Yaskawa INFORM job: test_long_tjr4.JBI

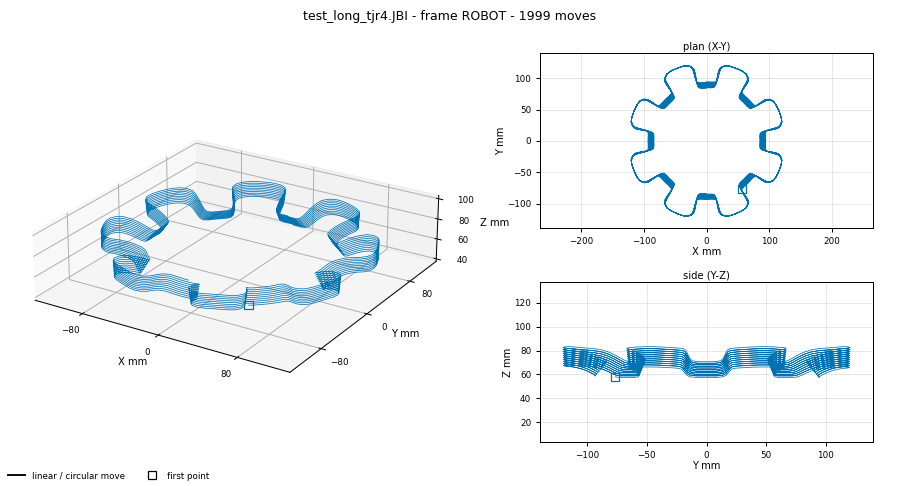
[picture p0: tool path of test_long_tjr4.JBI in frame ROBOT, 1999 of 2000 moves have a stored position in this frame; points joined in program order, loops and branches not executed]
version: 0
/JOB
//NAME test_long
//POS
///NPOS 48,0,0,2,0,0
///TOOL 1
///POSTYPE ROBOT
///RECTAN
///RCONF 1,0,0,0,0,0,0,0,0,0,0,0,0,0,0,0,0,0,0,0,0,0,0,0
C00000=56.550,-79.670,59.270,-0.1700,-0.0500,0.9800
C00001=57.060,-76.470,58.000,-0.5100,0.2200,0.8300
C00002=60.180,-72.990,57.500,-0.4400,0.4500,0.7800
C00003=63.630,-69.930,57.480,-0.4200,0.4700,0.7700
C00004=66.860,-66.860,57.500,-0.4500,0.4500,0.7700
C00005=69.930,-63.630,57.480,-0.4700,0.4200,0.7700
C00006=72.990,-60.180,57.500,-0.4500,0.4400,0.7800
C00007=76.470,-57.060,58.000,-0.2200,0.5100,0.8300
C00008=79.670,-56.550,59.270,0.0500,0.1700,0.9800
C00009=83.300,-57.850,61.030,-0.0000,-0.0000,1.0000
C00010=87.670,-60.190,62.880,-0.0400,-0.0700,1.0000
C00011=92.520,-62.920,64.320,-0.0600,-0.1100,0.9900
C00012=97.350,-65.090,65.040,-0.0300,-0.1200,0.9900
C00013=102.620,-64.760,65.430,0.0200,-0.0700,1.0000
C00014=107.590,-61.840,65.740,0.0300,-0.0300,1.0000
C00015=111.260,-56.800,66.060,0.0000,-0.0000,1.0000
C00016=114.160,-50.900,66.270,0.0000,-0.0000,1.0000
C00017=116.710,-44.730,66.270,0.0000,-0.0000,1.0000
C00018=118.840,-38.510,66.060,0.0000,-0.0000,1.0000
C00019=119.800,-32.350,65.740,0.0400,0.0000,1.0000
C00020=118.360,-26.770,65.430,0.0700,0.0300,1.0000
C00021=114.870,-22.810,65.040,0.0700,0.1000,0.9900
C00022=109.910,-20.930,64.320,0.0400,0.1200,0.9900
C00023=104.550,-19.430,62.880,0.0200,0.0800,1.0000
C00024=99.810,-18.000,61.030,0.0000,0.0000,1.0000
C00025=96.330,-16.350,59.270,-0.0800,-0.1500,0.9800
C00026=94.420,-13.720,58.000,-0.5100,-0.2000,0.8300
C00027=94.160,-9.060,57.500,-0.6300,0.0100,0.7800
C00028=94.440,-4.460,57.480,-0.6300,0.0300,0.7700
C00029=94.550,0.000,57.500,-0.6300,0.0000,0.7700
C00030=94.440,4.460,57.480,-0.6300,-0.0300,0.7700
C00031=94.160,9.060,57.500,-0.6300,-0.0100,0.7800
C00032=94.420,13.720,58.000,-0.5100,0.2000,0.8300
C00033=96.330,16.350,59.270,-0.0800,0.1500,0.9800
C00034=99.810,18.000,61.030,0.0000,-0.0000,1.0000
C00035=104.550,19.430,62.880,0.0200,-0.0800,1.0000
C00036=109.910,20.930,64.320,0.0400,-0.1200,0.9900
C00037=114.870,22.810,65.040,0.0700,-0.1000,0.9900
C00038=118.360,26.770,65.430,0.0700,-0.0300,1.0000
C00039=119.800,32.350,65.740,0.0400,-0.0000,1.0000
C00040=118.840,38.510,66.060,0.0000,0.0000,1.0000
C00041=116.710,44.730,66.270,0.0000,0.0000,1.0000
C00042=114.160,50.900,66.270,0.0000,0.0000,1.0000
C00043=111.260,56.800,66.060,0.0000,0.0000,1.0000
C00044=107.590,61.840,65.740,0.0300,0.0300,1.0000
C00045=102.620,64.760,65.430,0.0200,0.0700,1.0000
C00046=97.350,65.090,65.040,-0.0300,0.1200,0.9900
C00047=92.520,62.920,64.320,-0.0600,0.1100,0.9900
C00048=87.670,60.190,62.880,-0.0400,0.0700,1.0000
C00049=83.300,57.850,61.030,-0.0000,0.0000,1.0000
C00050=79.670,56.550,59.270,0.0500,-0.1700,0.9800
C00051=76.470,57.060,58.000,-0.2200,-0.5100,0.8300
C00052=72.990,60.180,57.500,-0.4500,-0.4400,0.7800
C00053=69.930,63.630,57.480,-0.4700,-0.4200,0.7700
C00054=66.860,66.860,57.500,-0.4500,-0.4500,0.7700
C00055=63.630,69.930,57.480,-0.4200,-0.4700,0.7700
C00056=60.180,72.990,57.500,-0.4400,-0.4500,0.7800
C00057=57.060,76.470,58.000,-0.5100,-0.2200,0.8300
C00058=56.550,79.670,59.270,-0.1700,0.0500,0.9800
C00059=57.850,83.300,61.030,0.0000,-0.0000,1.0000
C00060=60.190,87.670,62.880,0.0700,-0.0400,1.0000
C00061=62.920,92.520,64.320,0.1100,-0.0600,0.9900
C00062=65.090,97.350,65.040,0.1200,-0.0300,0.9900
C00063=64.760,102.620,65.430,0.0700,0.0200,1.0000
C00064=61.840,107.590,65.740,0.0300,0.0300,1.0000
C00065=56.800,111.260,66.060,0.0000,0.0000,1.0000
C00066=50.900,114.160,66.270,0.0000,0.0000,1.0000
C00067=44.730,116.710,66.270,0.0000,0.0000,1.0000
C00068=38.510,118.840,66.060,0.0000,0.0000,1.0000
C00069=32.350,119.800,65.740,-0.0000,0.0400,1.0000
C00070=26.770,118.360,65.430,-0.0300,0.0700,1.0000
C00071=22.810,114.870,65.040,-0.1000,0.0700,0.9900
C00072=20.930,109.910,64.320,-0.1200,0.0400,0.9900
C00073=19.430,104.550,62.880,-0.0800,0.0200,1.0000
C00074=18.000,99.810,61.030,-0.0000,0.0000,1.0000
C00075=16.350,96.330,59.270,0.1500,-0.0800,0.9800
C00076=13.720,94.420,58.000,0.2000,-0.5100,0.8300
C00077=9.060,94.160,57.500,-0.0100,-0.6300,0.7800
C00078=4.460,94.440,57.480,-0.0300,-0.6300,0.7700
C00079=0.000,94.550,57.500,0.0000,-0.6300,0.7700
C00080=0.000,93.470,58.810,0.0000,-0.6300,0.7700
C00081=4.360,93.370,58.800,-0.0300,-0.6300,0.7700
C00082=8.890,93.100,58.820,-0.0100,-0.6300,0.7800
C00083=13.520,93.390,59.340,0.2100,-0.5000,0.8400
C00084=16.100,95.380,60.660,0.1400,-0.0700,0.9900
C00085=17.710,99.000,62.500,-0.0100,0.0000,1.0000
C00086=19.110,103.930,64.430,-0.0800,0.0200,1.0000
C00087=20.580,109.500,65.930,-0.1200,0.0400,0.9900
C00088=22.440,114.660,66.690,-0.1100,0.0700,0.9900
C00089=26.420,118.310,67.090,-0.0400,0.0700,1.0000
C00090=32.070,119.850,67.420,-0.0000,0.0400,1.0000
C00091=38.330,118.900,67.750,0.0000,0.0000,1.0000
C00092=44.670,116.740,67.970,0.0000,0.0000,1.0000
C00093=50.960,114.130,67.970,0.0000,0.0000,1.0000
C00094=56.970,111.170,67.750,0.0000,0.0000,1.0000
C00095=62.070,107.420,67.420,0.0300,0.0300,1.0000
C00096=64.980,102.340,67.090,0.0700,0.0200,1.0000
C00097=65.210,96.940,66.690,0.1200,-0.0300,0.9900
C00098=62.880,91.990,65.930,0.1100,-0.0600,0.9900
C00099=59.970,87.000,64.430,0.0700,-0.0400,1.0000
C00100=57.480,82.530,62.500,0.0100,-0.0000,1.0000
C00101=56.060,78.830,60.660,-0.1500,0.0500,0.9900
C00102=56.480,75.600,59.340,-0.5100,-0.2100,0.8400
C00103=59.550,72.120,58.820,-0.4400,-0.4500,0.7800
C00104=62.940,69.100,58.800,-0.4200,-0.4700,0.7700
C00105=66.090,66.090,58.810,-0.4500,-0.4500,0.7700
C00106=69.100,62.940,58.800,-0.4700,-0.4200,0.7700
C00107=72.120,59.550,58.820,-0.4500,-0.4400,0.7800
C00108=75.600,56.480,59.340,-0.2100,-0.5100,0.8400
C00109=78.830,56.060,60.660,0.0500,-0.1500,0.9900
C00110=82.530,57.480,62.500,-0.0000,0.0100,1.0000
C00111=87.000,59.970,64.430,-0.0400,0.0700,1.0000
C00112=91.990,62.880,65.930,-0.0600,0.1100,0.9900
C00113=96.940,65.210,66.690,-0.0300,0.1200,0.9900
C00114=102.340,64.980,67.090,0.0200,0.0700,1.0000
C00115=107.420,62.070,67.420,0.0300,0.0300,1.0000
C00116=111.170,56.970,67.750,0.0000,0.0000,1.0000
C00117=114.130,50.960,67.970,0.0000,0.0000,1.0000
C00118=116.740,44.670,67.970,0.0000,0.0000,1.0000
C00119=118.900,38.330,67.750,0.0000,0.0000,1.0000
C00120=119.850,32.070,67.420,0.0400,-0.0000,1.0000
C00121=118.310,26.420,67.090,0.0700,-0.0400,1.0000
C00122=114.660,22.440,66.690,0.0700,-0.1100,0.9900
C00123=109.500,20.580,65.930,0.0400,-0.1200,0.9900
C00124=103.930,19.110,64.430,0.0200,-0.0800,1.0000
C00125=99.000,17.710,62.500,0.0000,-0.0100,1.0000
C00126=95.380,16.100,60.660,-0.0700,0.1400,0.9900
C00127=93.390,13.520,59.340,-0.5000,0.2100,0.8400
C00128=93.100,8.890,58.820,-0.6300,-0.0100,0.7800
C00129=93.370,4.360,58.800,-0.6300,-0.0300,0.7700
C00130=93.470,0.000,58.810,-0.6300,0.0000,0.7700
C00131=93.370,-4.360,58.800,-0.6300,0.0300,0.7700
C00132=93.100,-8.890,58.820,-0.6300,0.0100,0.7800
C00133=93.390,-13.520,59.340,-0.5000,-0.2100,0.8400
C00134=95.380,-16.100,60.660,-0.0700,-0.1400,0.9900
C00135=99.000,-17.710,62.500,0.0000,0.0100,1.0000
C00136=103.930,-19.110,64.430,0.0200,0.0800,1.0000
C00137=109.500,-20.580,65.930,0.0400,0.1200,0.9900
C00138=114.660,-22.440,66.690,0.0700,0.1100,0.9900
C00139=118.310,-26.420,67.090,0.0700,0.0400,1.0000
C00140=119.850,-32.070,67.420,0.0400,0.0000,1.0000
C00141=118.900,-38.330,67.750,0.0000,-0.0000,1.0000
C00142=116.740,-44.670,67.970,0.0000,-0.0000,1.0000
C00143=114.130,-50.960,67.970,0.0000,-0.0000,1.0000
C00144=111.170,-56.970,67.750,0.0000,-0.0000,1.0000
C00145=107.420,-62.070,67.420,0.0300,-0.0300,1.0000
C00146=102.340,-64.980,67.090,0.0200,-0.0700,1.0000
C00147=96.940,-65.210,66.690,-0.0300,-0.1200,0.9900
C00148=91.990,-62.880,65.930,-0.0600,-0.1100,0.9900
C00149=87.000,-59.970,64.430,-0.0400,-0.0700,1.0000
C00150=82.530,-57.480,62.500,-0.0000,-0.0100,1.0000
C00151=78.830,-56.060,60.660,0.0500,0.1500,0.9900
C00152=75.600,-56.480,59.340,-0.2100,0.5100,0.8400
C00153=72.120,-59.550,58.820,-0.4500,0.4400,0.7800
C00154=69.100,-62.940,58.800,-0.4700,0.4200,0.7700
C00155=66.090,-66.090,58.810,-0.4500,0.4500,0.7700
C00156=62.940,-69.100,58.800,-0.4200,0.4700,0.7700
C00157=59.550,-72.120,58.820,-0.4400,0.4500,0.7800
C00158=56.480,-75.600,59.340,-0.5100,0.2100,0.8400
C00159=56.060,-78.830,60.660,-0.1500,-0.0500,0.9900
C00160=57.480,-82.530,62.500,0.0100,0.0000,1.0000
C00161=59.970,-87.000,64.430,0.0700,0.0400,1.0000
C00162=62.880,-91.990,65.930,0.1100,0.0600,0.9900
C00163=65.210,-96.940,66.690,0.1200,0.0300,0.9900
C00164=64.980,-102.340,67.090,0.0700,-0.0200,1.0000
C00165=62.070,-107.420,67.420,0.0300,-0.0300,1.0000
C00166=56.970,-111.170,67.750,0.0000,-0.0000,1.0000
C00167=50.960,-114.130,67.970,0.0000,-0.0000,1.0000
C00168=44.670,-116.740,67.970,0.0000,-0.0000,1.0000
C00169=38.330,-118.900,67.750,0.0000,-0.0000,1.0000
C00170=32.070,-119.850,67.420,-0.0000,-0.0400,1.0000
C00171=26.420,-118.310,67.090,-0.0400,-0.0700,1.0000
C00172=22.440,-114.660,66.690,-0.1100,-0.0700,0.9900
C00173=20.580,-109.500,65.930,-0.1200,-0.0400,0.9900
C00174=19.110,-103.930,64.430,-0.0800,-0.0200,1.0000
C00175=17.710,-99.000,62.500,-0.0100,-0.0000,1.0000
C00176=16.100,-95.380,60.660,0.1400,0.0700,0.9900
C00177=13.520,-93.390,59.340,0.2100,0.5000,0.8400
C00178=8.890,-93.100,58.820,-0.0100,0.6300,0.7800
C00179=4.360,-93.370,58.800,-0.0300,0.6300,0.7700
C00180=0.000,-93.470,58.810,0.0000,0.6300,0.7700
C00181=0.000,-93.470,58.810,0.0000,0.6300,0.7700
C00182=-4.360,-93.370,58.800,0.0300,0.6300,0.7700
C00183=-8.890,-93.100,58.820,0.0100,0.6300,0.7800
C00184=-13.520,-93.390,59.340,-0.2100,0.5000,0.8400
C00185=-16.100,-95.380,60.660,-0.1400,0.0700,0.9900
C00186=-17.710,-99.000,62.500,0.0100,-0.0000,1.0000
C00187=-19.110,-103.930,64.430,0.0800,-0.0200,1.0000
C00188=-20.580,-109.500,65.930,0.1200,-0.0400,0.9900
C00189=-22.440,-114.660,66.690,0.1100,-0.0700,0.9900
C00190=-26.420,-118.310,67.090,0.0400,-0.0700,1.0000
C00191=-32.070,-119.850,67.420,0.0000,-0.0400,1.0000
C00192=-38.330,-118.900,67.750,-0.0000,-0.0000,1.0000
C00193=-44.670,-116.740,67.970,-0.0000,-0.0000,1.0000
C00194=-50.960,-114.130,67.970,-0.0000,-0.0000,1.0000
C00195=-56.970,-111.170,67.750,-0.0000,-0.0000,1.0000
C00196=-62.070,-107.420,67.420,-0.0300,-0.0300,1.0000
C00197=-64.980,-102.340,67.090,-0.0700,-0.0200,1.0000
C00198=-65.210,-96.940,66.690,-0.1200,0.0300,0.9900
C00199=-62.880,-91.990,65.930,-0.1100,0.0600,0.9900
C00200=-59.970,-87.000,64.430,-0.0700,0.0400,1.0000
C00201=-57.480,-82.530,62.500,-0.0100,0.0000,1.0000
C00202=-56.060,-78.830,60.660,0.1500,-0.0500,0.9900
C00203=-56.480,-75.600,59.340,0.5100,0.2100,0.8400
C00204=-59.550,-72.120,58.820,0.4400,0.4500,0.7800
C00205=-62.940,-69.100,58.800,0.4200,0.4700,0.7700
C00206=-66.090,-66.090,58.810,0.4500,0.4500,0.7700
C00207=-69.100,-62.940,58.800,0.4700,0.4200,0.7700
C00208=-72.120,-59.550,58.820,0.4500,0.4400,0.7800
C00209=-75.600,-56.480,59.340,0.2100,0.5100,0.8400
C00210=-78.830,-56.060,60.660,-0.0500,0.1500,0.9900
C00211=-82.530,-57.480,62.500,0.0000,-0.0100,1.0000
C00212=-87.000,-59.970,64.430,0.0400,-0.0700,1.0000
C00213=-91.990,-62.880,65.930,0.0600,-0.1100,0.9900
C00214=-96.940,-65.210,66.690,0.0300,-0.1200,0.9900
C00215=-102.340,-64.980,67.090,-0.0200,-0.0700,1.0000
C00216=-107.420,-62.070,67.420,-0.0300,-0.0300,1.0000
C00217=-111.170,-56.970,67.750,-0.0000,-0.0000,1.0000
C00218=-114.130,-50.960,67.970,-0.0000,-0.0000,1.0000
C00219=-116.740,-44.670,67.970,-0.0000,-0.0000,1.0000
C00220=-118.900,-38.330,67.750,-0.0000,-0.0000,1.0000
C00221=-119.850,-32.070,67.420,-0.0400,0.0000,1.0000
C00222=-118.310,-26.420,67.090,-0.0700,0.0400,1.0000
C00223=-114.660,-22.440,66.690,-0.0700,0.1100,0.9900
C00224=-109.500,-20.580,65.930,-0.0400,0.1200,0.9900
C00225=-103.930,-19.110,64.430,-0.0200,0.0800,1.0000
C00226=-99.000,-17.710,62.500,-0.0000,0.0100,1.0000
C00227=-95.380,-16.100,60.660,0.0700,-0.1400,0.9900
C00228=-93.390,-13.520,59.340,0.5000,-0.2100,0.8400
C00229=-93.100,-8.890,58.820,0.6300,0.0100,0.7800
C00230=-93.370,-4.360,58.800,0.6300,0.0300,0.7700
C00231=-93.470,0.000,58.810,0.6300,-0.0000,0.7700
C00232=-93.370,4.360,58.800,0.6300,-0.0300,0.7700
C00233=-93.100,8.890,58.820,0.6300,-0.0100,0.7800
C00234=-93.390,13.520,59.340,0.5000,0.2100,0.8400
C00235=-95.380,16.100,60.660,0.0700,0.1400,0.9900
C00236=-99.000,17.710,62.500,-0.0000,-0.0100,1.0000
C00237=-103.930,19.110,64.430,-0.0200,-0.0800,1.0000
C00238=-109.500,20.580,65.930,-0.0400,-0.1200,0.9900
C00239=-114.660,22.440,66.690,-0.0700,-0.1100,0.9900
C00240=-118.310,26.420,67.090,-0.0700,-0.0400,1.0000
C00241=-119.850,32.070,67.420,-0.0400,-0.0000,1.0000
C00242=-118.900,38.330,67.750,-0.0000,0.0000,1.0000
C00243=-116.740,44.670,67.970,-0.0000,0.0000,1.0000
C00244=-114.130,50.960,67.970,-0.0000,0.0000,1.0000
C00245=-111.170,56.970,67.750,-0.0000,0.0000,1.0000
C00246=-107.420,62.070,67.420,-0.0300,0.0300,1.0000
C00247=-102.340,64.980,67.090,-0.0200,0.0700,1.0000
C00248=-96.940,65.210,66.690,0.0300,0.1200,0.9900
C00249=-91.990,62.880,65.930,0.0600,0.1100,0.9900
C00250=-87.000,59.970,64.430,0.0400,0.0700,1.0000
C00251=-82.530,57.480,62.500,0.0000,0.0100,1.0000
C00252=-78.830,56.060,60.660,-0.0500,-0.1500,0.9900
C00253=-75.600,56.480,59.340,0.2100,-0.5100,0.8400
C00254=-72.120,59.550,58.820,0.4500,-0.4400,0.7800
C00255=-69.100,62.940,58.800,0.4700,-0.4200,0.7700
C00256=-66.090,66.090,58.810,0.4500,-0.4500,0.7700
C00257=-62.940,69.100,58.800,0.4200,-0.4700,0.7700
C00258=-59.550,72.120,58.820,0.4400,-0.4500,0.7800
C00259=-56.480,75.600,59.340,0.5100,-0.2100,0.8400
C00260=-56.060,78.830,60.660,0.1500,0.0500,0.9900
C00261=-57.480,82.530,62.500,-0.0100,-0.0000,1.0000
C00262=-59.970,87.000,64.430,-0.0700,-0.0400,1.0000
C00263=-62.880,91.990,65.930,-0.1100,-0.0600,0.9900
C00264=-65.210,96.940,66.690,-0.1200,-0.0300,0.9900
C00265=-64.980,102.340,67.090,-0.0700,0.0200,1.0000
C00266=-62.070,107.420,67.420,-0.0300,0.0300,1.0000
C00267=-56.970,111.170,67.750,-0.0000,0.0000,1.0000
C00268=-50.960,114.130,67.970,-0.0000,0.0000,1.0000
C00269=-44.670,116.740,67.970,-0.0000,0.0000,1.0000
C00270=-38.330,118.900,67.750,-0.0000,0.0000,1.0000
C00271=-32.070,119.850,67.420,0.0000,0.0400,1.0000
C00272=-26.420,118.310,67.090,0.0400,0.0700,1.0000
C00273=-22.440,114.660,66.690,0.1100,0.0700,0.9900
C00274=-20.580,109.500,65.930,0.1200,0.0400,0.9900
C00275=-19.110,103.930,64.430,0.0800,0.0200,1.0000
C00276=-17.710,99.000,62.500,0.0100,0.0000,1.0000
C00277=-16.100,95.380,60.660,-0.1400,-0.0700,0.9900
C00278=-13.520,93.390,59.340,-0.2100,-0.5000,0.8400
C00279=-8.890,93.100,58.820,0.0100,-0.6300,0.7800
C00280=-4.360,93.370,58.800,0.0300,-0.6300,0.7700
C00281=0.000,93.470,58.810,0.0000,-0.6300,0.7700
C00282=0.000,92.400,60.130,-0.0000,-0.6300,0.7700
C00283=-4.260,92.300,60.110,0.0300,-0.6300,0.7700
C00284=-8.720,92.040,60.140,0.0000,-0.6300,0.7800
C00285=-13.320,92.360,60.680,-0.2200,-0.5000,0.8400
C00286=-15.850,94.440,62.050,-0.1300,-0.0600,0.9900
C00287=-17.420,98.200,63.970,0.0200,0.0100,1.0000
C00288=-18.790,103.310,65.980,0.0900,0.0200,1.0000
C00289=-20.240,109.100,67.550,0.1200,0.0400,0.9900
C00290=-22.060,114.460,68.330,0.1100,0.0700,0.9900
C00291=-26.060,118.270,68.750,0.0400,0.0700,1.0000
C00292=-31.790,119.900,69.090,0.0000,0.0400,1.0000
C00293=-38.150,118.960,69.440,-0.0000,0.0000,1.0000
C00294=-44.610,116.760,69.670,-0.0000,0.0000,1.0000
C00295=-51.020,114.110,69.670,-0.0000,0.0000,1.0000
C00296=-57.140,111.090,69.440,-0.0000,0.0000,1.0000
C00297=-62.310,107.260,69.090,-0.0300,0.0300,1.0000
C00298=-65.200,102.060,68.750,-0.0800,0.0200,1.0000
C00299=-65.330,96.530,68.330,-0.1300,-0.0300,0.9900
C00300=-62.830,91.460,67.550,-0.1100,-0.0600,0.9900
C00301=-59.760,86.340,65.980,-0.0800,-0.0400,1.0000
C00302=-57.120,81.750,63.970,-0.0200,-0.0100,1.0000
C00303=-55.570,77.990,62.050,0.1300,0.0400,0.9900
C00304=-55.890,74.730,60.680,0.5000,-0.2000,0.8400
C00305=-58.910,71.250,60.140,0.4400,-0.4500,0.7800
C00306=-62.250,68.280,60.110,0.4200,-0.4700,0.7700
C00307=-65.330,65.330,60.130,0.4500,-0.4500,0.7700
C00308=-68.280,62.250,60.110,0.4700,-0.4200,0.7700
C00309=-71.250,58.910,60.140,0.4500,-0.4400,0.7800
C00310=-74.730,55.890,60.680,0.2000,-0.5000,0.8400
C00311=-77.990,55.570,62.050,-0.0400,-0.1300,0.9900
C00312=-81.750,57.120,63.970,0.0100,0.0200,1.0000
C00313=-86.340,59.760,65.980,0.0400,0.0800,1.0000
C00314=-91.460,62.830,67.550,0.0600,0.1100,0.9900
C00315=-96.530,65.330,68.330,0.0300,0.1300,0.9900
C00316=-102.060,65.200,68.750,-0.0200,0.0800,1.0000
C00317=-107.260,62.310,69.090,-0.0300,0.0300,1.0000
C00318=-111.090,57.140,69.440,-0.0000,0.0000,1.0000
C00319=-114.110,51.020,69.670,-0.0000,0.0000,1.0000
C00320=-116.760,44.610,69.670,-0.0000,0.0000,1.0000
C00321=-118.960,38.150,69.440,-0.0000,0.0000,1.0000
C00322=-119.900,31.790,69.090,-0.0400,-0.0000,1.0000
C00323=-118.270,26.060,68.750,-0.0700,-0.0400,1.0000
C00324=-114.460,22.060,68.330,-0.0700,-0.1100,0.9900
C00325=-109.100,20.240,67.550,-0.0400,-0.1200,0.9900
C00326=-103.310,18.790,65.980,-0.0200,-0.0900,1.0000
C00327=-98.200,17.420,63.970,-0.0100,-0.0200,1.0000
C00328=-94.440,15.850,62.050,0.0600,0.1300,0.9900
C00329=-92.360,13.320,60.680,0.5000,0.2200,0.8400
C00330=-92.040,8.720,60.140,0.6300,-0.0000,0.7800
C00331=-92.300,4.260,60.110,0.6300,-0.0300,0.7700
C00332=-92.400,0.000,60.130,0.6300,0.0000,0.7700
C00333=-92.300,-4.260,60.110,0.6300,0.0300,0.7700
C00334=-92.040,-8.720,60.140,0.6300,0.0000,0.7800
C00335=-92.360,-13.320,60.680,0.5000,-0.2200,0.8400
C00336=-94.440,-15.850,62.050,0.0600,-0.1300,0.9900
C00337=-98.200,-17.420,63.970,-0.0100,0.0200,1.0000
C00338=-103.310,-18.790,65.980,-0.0200,0.0900,1.0000
C00339=-109.100,-20.240,67.550,-0.0400,0.1200,0.9900
C00340=-114.460,-22.060,68.330,-0.0700,0.1100,0.9900
C00341=-118.270,-26.060,68.750,-0.0700,0.0400,1.0000
C00342=-119.900,-31.790,69.090,-0.0400,0.0000,1.0000
C00343=-118.960,-38.150,69.440,-0.0000,-0.0000,1.0000
C00344=-116.760,-44.610,69.670,-0.0000,-0.0000,1.0000
C00345=-114.110,-51.020,69.670,-0.0000,-0.0000,1.0000
C00346=-111.090,-57.140,69.440,-0.0000,-0.0000,1.0000
C00347=-107.260,-62.310,69.090,-0.0300,-0.0300,1.0000
C00348=-102.060,-65.200,68.750,-0.0200,-0.0800,1.0000
C00349=-96.530,-65.330,68.330,0.0300,-0.1300,0.9900
C00350=-91.460,-62.830,67.550,0.0600,-0.1100,0.9900
C00351=-86.340,-59.760,65.980,0.0400,-0.0800,1.0000
C00352=-81.750,-57.120,63.970,0.0100,-0.0200,1.0000
C00353=-77.990,-55.570,62.050,-0.0400,0.1300,0.9900
C00354=-74.730,-55.890,60.680,0.2000,0.5000,0.8400
C00355=-71.250,-58.910,60.140,0.4500,0.4400,0.7800
C00356=-68.280,-62.250,60.110,0.4700,0.4200,0.7700
C00357=-65.330,-65.330,60.130,0.4500,0.4500,0.7700
C00358=-62.250,-68.280,60.110,0.4200,0.4700,0.7700
C00359=-58.910,-71.250,60.140,0.4400,0.4500,0.7800
C00360=-55.890,-74.730,60.680,0.5000,0.2000,0.8400
C00361=-55.570,-77.990,62.050,0.1300,-0.0400,0.9900
C00362=-57.120,-81.750,63.970,-0.0200,0.0100,1.0000
C00363=-59.760,-86.340,65.980,-0.0800,0.0400,1.0000
C00364=-62.830,-91.460,67.550,-0.1100,0.0600,0.9900
C00365=-65.330,-96.530,68.330,-0.1300,0.0300,0.9900
C00366=-65.200,-102.060,68.750,-0.0800,-0.0200,1.0000
C00367=-62.310,-107.260,69.090,-0.0300,-0.0300,1.0000
C00368=-57.140,-111.090,69.440,-0.0000,-0.0000,1.0000
C00369=-51.020,-114.110,69.670,-0.0000,-0.0000,1.0000
C00370=-44.610,-116.760,69.670,-0.0000,-0.0000,1.0000
C00371=-38.150,-118.960,69.440,-0.0000,-0.0000,1.0000
C00372=-31.790,-119.900,69.090,0.0000,-0.0400,1.0000
C00373=-26.060,-118.270,68.750,0.0400,-0.0700,1.0000
C00374=-22.060,-114.460,68.330,0.1100,-0.0700,0.9900
C00375=-20.240,-109.100,67.550,0.1200,-0.0400,0.9900
C00376=-18.790,-103.310,65.980,0.0900,-0.0200,1.0000
C00377=-17.420,-98.200,63.970,0.0200,-0.0100,1.0000
C00378=-15.850,-94.440,62.050,-0.1300,0.0600,0.9900
C00379=-13.320,-92.360,60.680,-0.2200,0.5000,0.8400
C00380=-8.720,-92.040,60.140,0.0000,0.6300,0.7800
C00381=-4.260,-92.300,60.110,0.0300,0.6300,0.7700
C00382=0.000,-92.400,60.130,-0.0000,0.6300,0.7700
C00383=0.000,-92.400,60.130,-0.0000,0.6300,0.7700
C00384=4.260,-92.300,60.110,-0.0300,0.6300,0.7700
C00385=8.720,-92.040,60.140,-0.0000,0.6300,0.7800
C00386=13.320,-92.360,60.680,0.2200,0.5000,0.8400
C00387=15.850,-94.440,62.050,0.1300,0.0600,0.9900
C00388=17.420,-98.200,63.970,-0.0200,-0.0100,1.0000
C00389=18.790,-103.310,65.980,-0.0900,-0.0200,1.0000
C00390=20.240,-109.100,67.550,-0.1200,-0.0400,0.9900
C00391=22.060,-114.460,68.330,-0.1100,-0.0700,0.9900
C00392=26.060,-118.270,68.750,-0.0400,-0.0700,1.0000
C00393=31.790,-119.900,69.090,-0.0000,-0.0400,1.0000
C00394=38.150,-118.960,69.440,0.0000,-0.0000,1.0000
C00395=44.610,-116.760,69.670,0.0000,-0.0000,1.0000
C00396=51.020,-114.110,69.670,0.0000,-0.0000,1.0000
C00397=57.140,-111.090,69.440,0.0000,-0.0000,1.0000
C00398=62.310,-107.260,69.090,0.0300,-0.0300,1.0000
C00399=65.200,-102.060,68.750,0.0800,-0.0200,1.0000
C00400=65.330,-96.530,68.330,0.1300,0.0300,0.9900
C00401=62.830,-91.460,67.550,0.1100,0.0600,0.9900
C00402=59.760,-86.340,65.980,0.0800,0.0400,1.0000
C00403=57.120,-81.750,63.970,0.0200,0.0100,1.0000
C00404=55.570,-77.990,62.050,-0.1300,-0.0400,0.9900
C00405=55.890,-74.730,60.680,-0.5000,0.2000,0.8400
C00406=58.910,-71.250,60.140,-0.4400,0.4500,0.7800
C00407=62.250,-68.280,60.110,-0.4200,0.4700,0.7700
C00408=65.330,-65.330,60.130,-0.4500,0.4500,0.7700
C00409=68.280,-62.250,60.110,-0.4700,0.4200,0.7700
C00410=71.250,-58.910,60.140,-0.4500,0.4400,0.7800
C00411=74.730,-55.890,60.680,-0.2000,0.5000,0.8400
C00412=77.990,-55.570,62.050,0.0400,0.1300,0.9900
C00413=81.750,-57.120,63.970,-0.0100,-0.0200,1.0000
C00414=86.340,-59.760,65.980,-0.0400,-0.0800,1.0000
C00415=91.460,-62.830,67.550,-0.0600,-0.1100,0.9900
C00416=96.530,-65.330,68.330,-0.0300,-0.1300,0.9900
C00417=102.060,-65.200,68.750,0.0200,-0.0800,1.0000
C00418=107.260,-62.310,69.090,0.0300,-0.0300,1.0000
C00419=111.090,-57.140,69.440,0.0000,-0.0000,1.0000
C00420=114.110,-51.020,69.670,0.0000,-0.0000,1.0000
C00421=116.760,-44.610,69.670,0.0000,-0.0000,1.0000
C00422=118.960,-38.150,69.440,0.0000,-0.0000,1.0000
C00423=119.900,-31.790,69.090,0.0400,0.0000,1.0000
C00424=118.270,-26.060,68.750,0.0700,0.0400,1.0000
C00425=114.460,-22.060,68.330,0.0700,0.1100,0.9900
C00426=109.100,-20.240,67.550,0.0400,0.1200,0.9900
C00427=103.310,-18.790,65.980,0.0200,0.0900,1.0000
C00428=98.200,-17.420,63.970,0.0100,0.0200,1.0000
C00429=94.440,-15.850,62.050,-0.0600,-0.1300,0.9900
C00430=92.360,-13.320,60.680,-0.5000,-0.2200,0.8400
C00431=92.040,-8.720,60.140,-0.6300,0.0000,0.7800
C00432=92.300,-4.260,60.110,-0.6300,0.0300,0.7700
C00433=92.400,0.000,60.130,-0.6300,-0.0000,0.7700
C00434=92.300,4.260,60.110,-0.6300,-0.0300,0.7700
C00435=92.040,8.720,60.140,-0.6300,-0.0000,0.7800
C00436=92.360,13.320,60.680,-0.5000,0.2200,0.8400
C00437=94.440,15.850,62.050,-0.0600,0.1300,0.9900
C00438=98.200,17.420,63.970,0.0100,-0.0200,1.0000
C00439=103.310,18.790,65.980,0.0200,-0.0900,1.0000
C00440=109.100,20.240,67.550,0.0400,-0.1200,0.9900
C00441=114.460,22.060,68.330,0.0700,-0.1100,0.9900
C00442=118.270,26.060,68.750,0.0700,-0.0400,1.0000
C00443=119.900,31.790,69.090,0.0400,-0.0000,1.0000
C00444=118.960,38.150,69.440,0.0000,0.0000,1.0000
C00445=116.760,44.610,69.670,0.0000,0.0000,1.0000
C00446=114.110,51.020,69.670,0.0000,0.0000,1.0000
C00447=111.090,57.140,69.440,0.0000,0.0000,1.0000
C00448=107.260,62.310,69.090,0.0300,0.0300,1.0000
C00449=102.060,65.200,68.750,0.0200,0.0800,1.0000
C00450=96.530,65.330,68.330,-0.0300,0.1300,0.9900
C00451=91.460,62.830,67.550,-0.0600,0.1100,0.9900
C00452=86.340,59.760,65.980,-0.0400,0.0800,1.0000
C00453=81.750,57.120,63.970,-0.0100,0.0200,1.0000
C00454=77.990,55.570,62.050,0.0400,-0.1300,0.9900
C00455=74.730,55.890,60.680,-0.2000,-0.5000,0.8400
C00456=71.250,58.910,60.140,-0.4500,-0.4400,0.7800
C00457=68.280,62.250,60.110,-0.4700,-0.4200,0.7700
C00458=65.330,65.330,60.130,-0.4500,-0.4500,0.7700
C00459=62.250,68.280,60.110,-0.4200,-0.4700,0.7700
C00460=58.910,71.250,60.140,-0.4400,-0.4500,0.7800
C00461=55.890,74.730,60.680,-0.5000,-0.2000,0.8400
C00462=55.570,77.990,62.050,-0.1300,0.0400,0.9900
C00463=57.120,81.750,63.970,0.0200,-0.0100,1.0000
C00464=59.760,86.340,65.980,0.0800,-0.0400,1.0000
C00465=62.830,91.460,67.550,0.1100,-0.0600,0.9900
C00466=65.330,96.530,68.330,0.1300,-0.0300,0.9900
C00467=65.200,102.060,68.750,0.0800,0.0200,1.0000
C00468=62.310,107.260,69.090,0.0300,0.0300,1.0000
C00469=57.140,111.090,69.440,0.0000,0.0000,1.0000
C00470=51.020,114.110,69.670,0.0000,0.0000,1.0000
C00471=44.610,116.760,69.670,0.0000,0.0000,1.0000
C00472=38.150,118.960,69.440,0.0000,0.0000,1.0000
C00473=31.790,119.900,69.090,-0.0000,0.0400,1.0000
C00474=26.060,118.270,68.750,-0.0400,0.0700,1.0000
C00475=22.060,114.460,68.330,-0.1100,0.0700,0.9900
C00476=20.240,109.100,67.550,-0.1200,0.0400,0.9900
C00477=18.790,103.310,65.980,-0.0900,0.0200,1.0000
C00478=17.420,98.200,63.970,-0.0200,0.0100,1.0000
C00479=15.850,94.440,62.050,0.1300,-0.0600,0.9900
C00480=13.320,92.360,60.680,0.2200,-0.5000,0.8400
C00481=8.720,92.040,60.140,-0.0000,-0.6300,0.7800
C00482=4.260,92.300,60.110,-0.0300,-0.6300,0.7700
C00483=0.000,92.400,60.130,-0.0000,-0.6300,0.7700
C00484=0.000,91.320,61.440,-0.0000,-0.6300,0.7700
C00485=4.160,91.220,61.430,-0.0300,-0.6300,0.7700
C00486=8.560,90.970,61.450,-0.0000,-0.6300,0.7800
C00487=13.120,91.330,62.020,0.2300,-0.4900,0.8400
C00488=15.600,93.500,63.440,0.1100,-0.0500,0.9900
C00489=17.130,97.400,65.440,-0.0200,0.0100,1.0000
C00490=18.480,102.690,67.530,-0.0900,0.0200,1.0000
C00491=19.900,108.690,69.160,-0.1300,0.0400,0.9900
C00492=21.690,114.260,69.980,-0.1200,0.0700,0.9900
C00493=25.720,118.230,70.410,-0.0400,0.0700,1.0000
C00494=31.510,119.950,70.770,-0.0000,0.0400,1.0000
C00495=37.980,119.010,71.130,0.0000,0.0000,1.0000
C00496=44.550,116.780,71.370,0.0000,0.0000,1.0000
C00497=51.070,114.080,71.370,0.0000,0.0000,1.0000
C00498=57.300,111.010,71.130,0.0000,0.0000,1.0000
C00499=62.540,107.100,70.770,0.0300,0.0300,1.0000
C00500=65.420,101.780,70.410,0.0800,0.0200,1.0000
C00501=65.450,96.130,69.980,0.1300,-0.0400,0.9900
C00502=62.780,90.930,69.160,0.1200,-0.0600,0.9900
C00503=59.550,85.680,67.530,0.0800,-0.0500,1.0000
C00504=56.760,80.980,65.440,0.0200,-0.0100,1.0000
C00505=55.080,77.140,63.440,-0.1200,0.0400,0.9900
C00506=55.310,73.860,62.020,-0.5000,-0.1800,0.8400
C00507=58.280,70.380,61.450,-0.4400,-0.4400,0.7800
C00508=61.560,67.450,61.430,-0.4200,-0.4700,0.7700
C00509=64.570,64.570,61.440,-0.4500,-0.4500,0.7700
C00510=67.450,61.560,61.430,-0.4700,-0.4200,0.7700
C00511=70.380,58.280,61.450,-0.4400,-0.4400,0.7800
C00512=73.860,55.310,62.020,-0.1800,-0.5000,0.8400
C00513=77.140,55.080,63.440,0.0400,-0.1200,0.9900
C00514=80.980,56.760,65.440,-0.0100,0.0200,1.0000
C00515=85.680,59.550,67.530,-0.0500,0.0800,1.0000
C00516=90.930,62.780,69.160,-0.0600,0.1200,0.9900
C00517=96.130,65.450,69.980,-0.0400,0.1300,0.9900
C00518=101.780,65.420,70.410,0.0200,0.0800,1.0000
C00519=107.100,62.540,70.770,0.0300,0.0300,1.0000
C00520=111.010,57.300,71.130,0.0000,0.0000,1.0000
C00521=114.080,51.070,71.370,0.0000,0.0000,1.0000
C00522=116.780,44.550,71.370,0.0000,0.0000,1.0000
C00523=119.010,37.980,71.130,0.0000,0.0000,1.0000
C00524=119.950,31.510,70.770,0.0400,-0.0000,1.0000
C00525=118.230,25.720,70.410,0.0700,-0.0400,1.0000
C00526=114.260,21.690,69.980,0.0700,-0.1200,0.9900
C00527=108.690,19.900,69.160,0.0400,-0.1300,0.9900
C00528=102.690,18.480,67.530,0.0200,-0.0900,1.0000
C00529=97.400,17.130,65.440,0.0100,-0.0200,1.0000
C00530=93.500,15.600,63.440,-0.0500,0.1100,0.9900
C00531=91.330,13.120,62.020,-0.4900,0.2300,0.8400
C00532=90.970,8.560,61.450,-0.6300,-0.0000,0.7800
C00533=91.220,4.160,61.430,-0.6300,-0.0300,0.7700
C00534=91.320,0.000,61.440,-0.6300,-0.0000,0.7700
C00535=91.220,-4.160,61.430,-0.6300,0.0300,0.7700
C00536=90.970,-8.560,61.450,-0.6300,0.0000,0.7800
C00537=91.330,-13.120,62.020,-0.4900,-0.2300,0.8400
C00538=93.500,-15.600,63.440,-0.0500,-0.1100,0.9900
C00539=97.400,-17.130,65.440,0.0100,0.0200,1.0000
C00540=102.690,-18.480,67.530,0.0200,0.0900,1.0000
C00541=108.690,-19.900,69.160,0.0400,0.1300,0.9900
C00542=114.260,-21.690,69.980,0.0700,0.1200,0.9900
C00543=118.230,-25.720,70.410,0.0700,0.0400,1.0000
C00544=119.950,-31.510,70.770,0.0400,0.0000,1.0000
C00545=119.010,-37.980,71.130,0.0000,-0.0000,1.0000
C00546=116.780,-44.550,71.370,0.0000,-0.0000,1.0000
C00547=114.080,-51.070,71.370,0.0000,-0.0000,1.0000
C00548=111.010,-57.300,71.130,0.0000,-0.0000,1.0000
C00549=107.100,-62.540,70.770,0.0300,-0.0300,1.0000
C00550=101.780,-65.420,70.410,0.0200,-0.0800,1.0000
C00551=96.130,-65.450,69.980,-0.0400,-0.1300,0.9900
C00552=90.930,-62.780,69.160,-0.0600,-0.1200,0.9900
C00553=85.680,-59.550,67.530,-0.0500,-0.0800,1.0000
C00554=80.980,-56.760,65.440,-0.0100,-0.0200,1.0000
C00555=77.140,-55.080,63.440,0.0400,0.1200,0.9900
C00556=73.860,-55.310,62.020,-0.1800,0.5000,0.8400
C00557=70.380,-58.280,61.450,-0.4400,0.4400,0.7800
C00558=67.450,-61.560,61.430,-0.4700,0.4200,0.7700
C00559=64.570,-64.570,61.440,-0.4500,0.4500,0.7700
C00560=61.560,-67.450,61.430,-0.4200,0.4700,0.7700
C00561=58.280,-70.380,61.450,-0.4400,0.4400,0.7800
C00562=55.310,-73.860,62.020,-0.5000,0.1800,0.8400
C00563=55.080,-77.140,63.440,-0.1200,-0.0400,0.9900
C00564=56.760,-80.980,65.440,0.0200,0.0100,1.0000
C00565=59.550,-85.680,67.530,0.0800,0.0500,1.0000
C00566=62.780,-90.930,69.160,0.1200,0.0600,0.9900
C00567=65.450,-96.130,69.980,0.1300,0.0400,0.9900
C00568=65.420,-101.780,70.410,0.0800,-0.0200,1.0000
C00569=62.540,-107.100,70.770,0.0300,-0.0300,1.0000
C00570=57.300,-111.010,71.130,0.0000,-0.0000,1.0000
C00571=51.070,-114.080,71.370,0.0000,-0.0000,1.0000
C00572=44.550,-116.780,71.370,0.0000,-0.0000,1.0000
C00573=37.980,-119.010,71.130,0.0000,-0.0000,1.0000
C00574=31.510,-119.950,70.770,-0.0000,-0.0400,1.0000
C00575=25.720,-118.230,70.410,-0.0400,-0.0700,1.0000
C00576=21.690,-114.260,69.980,-0.1200,-0.0700,0.9900
C00577=19.900,-108.690,69.160,-0.1300,-0.0400,0.9900
C00578=18.480,-102.690,67.530,-0.0900,-0.0200,1.0000
C00579=17.130,-97.400,65.440,-0.0200,-0.0100,1.0000
C00580=15.600,-93.500,63.440,0.1100,0.0500,0.9900
C00581=13.120,-91.330,62.020,0.2300,0.4900,0.8400
C00582=8.560,-90.970,61.450,-0.0000,0.6300,0.7800
C00583=4.160,-91.220,61.430,-0.0300,0.6300,0.7700
C00584=0.000,-91.320,61.440,-0.0000,0.6300,0.7700
C00585=0.000,-91.320,61.440,-0.0000,0.6300,0.7700
C00586=-4.160,-91.220,61.430,0.0300,0.6300,0.7700
C00587=-8.560,-90.970,61.450,0.0000,0.6300,0.7800
C00588=-13.120,-91.330,62.020,-0.2300,0.4900,0.8400
C00589=-15.600,-93.500,63.440,-0.1100,0.0500,0.9900
C00590=-17.130,-97.400,65.440,0.0200,-0.0100,1.0000
C00591=-18.480,-102.690,67.530,0.0900,-0.0200,1.0000
C00592=-19.900,-108.690,69.160,0.1300,-0.0400,0.9900
C00593=-21.690,-114.260,69.980,0.1200,-0.0700,0.9900
C00594=-25.720,-118.230,70.410,0.0400,-0.0700,1.0000
C00595=-31.510,-119.950,70.770,0.0000,-0.0400,1.0000
C00596=-37.980,-119.010,71.130,-0.0000,-0.0000,1.0000
C00597=-44.550,-116.780,71.370,-0.0000,-0.0000,1.0000
C00598=-51.070,-114.080,71.370,-0.0000,-0.0000,1.0000
C00599=-57.300,-111.010,71.130,-0.0000,-0.0000,1.0000
C00600=-62.540,-107.100,70.770,-0.0300,-0.0300,1.0000
C00601=-65.420,-101.780,70.410,-0.0800,-0.0200,1.0000
C00602=-65.450,-96.130,69.980,-0.1300,0.0400,0.9900
C00603=-62.780,-90.930,69.160,-0.1200,0.0600,0.9900
C00604=-59.550,-85.680,67.530,-0.0800,0.0500,1.0000
C00605=-56.760,-80.980,65.440,-0.0200,0.0100,1.0000
C00606=-55.080,-77.140,63.440,0.1200,-0.0400,0.9900
C00607=-55.310,-73.860,62.020,0.5000,0.1800,0.8400
C00608=-58.280,-70.380,61.450,0.4400,0.4400,0.7800
C00609=-61.560,-67.450,61.430,0.4200,0.4700,0.7700
C00610=-64.570,-64.570,61.440,0.4500,0.4500,0.7700
C00611=-67.450,-61.560,61.430,0.4700,0.4200,0.7700
C00612=-70.380,-58.280,61.450,0.4400,0.4400,0.7800
C00613=-73.860,-55.310,62.020,0.1800,0.5000,0.8400
C00614=-77.140,-55.080,63.440,-0.0400,0.1200,0.9900
C00615=-80.980,-56.760,65.440,0.0100,-0.0200,1.0000
C00616=-85.680,-59.550,67.530,0.0500,-0.0800,1.0000
C00617=-90.930,-62.780,69.160,0.0600,-0.1200,0.9900
C00618=-96.130,-65.450,69.980,0.0400,-0.1300,0.9900
C00619=-101.780,-65.420,70.410,-0.0200,-0.0800,1.0000
C00620=-107.100,-62.540,70.770,-0.0300,-0.0300,1.0000
C00621=-111.010,-57.300,71.130,-0.0000,-0.0000,1.0000
C00622=-114.080,-51.070,71.370,-0.0000,-0.0000,1.0000
C00623=-116.780,-44.550,71.370,-0.0000,-0.0000,1.0000
C00624=-119.010,-37.980,71.130,-0.0000,-0.0000,1.0000
C00625=-119.950,-31.510,70.770,-0.0400,0.0000,1.0000
C00626=-118.230,-25.720,70.410,-0.0700,0.0400,1.0000
C00627=-114.260,-21.690,69.980,-0.0700,0.1200,0.9900
C00628=-108.690,-19.900,69.160,-0.0400,0.1300,0.9900
C00629=-102.690,-18.480,67.530,-0.0200,0.0900,1.0000
C00630=-97.400,-17.130,65.440,-0.0100,0.0200,1.0000
C00631=-93.500,-15.600,63.440,0.0500,-0.1100,0.9900
C00632=-91.330,-13.120,62.020,0.4900,-0.2300,0.8400
C00633=-90.970,-8.560,61.450,0.6300,0.0000,0.7800
C00634=-91.220,-4.160,61.430,0.6300,0.0300,0.7700
C00635=-91.320,0.000,61.440,0.6300,0.0000,0.7700
C00636=-91.220,4.160,61.430,0.6300,-0.0300,0.7700
C00637=-90.970,8.560,61.450,0.6300,-0.0000,0.7800
C00638=-91.330,13.120,62.020,0.4900,0.2300,0.8400
C00639=-93.500,15.600,63.440,0.0500,0.1100,0.9900
C00640=-97.400,17.130,65.440,-0.0100,-0.0200,1.0000
C00641=-102.690,18.480,67.530,-0.0200,-0.0900,1.0000
C00642=-108.690,19.900,69.160,-0.0400,-0.1300,0.9900
C00643=-114.260,21.690,69.980,-0.0700,-0.1200,0.9900
C00644=-118.230,25.720,70.410,-0.0700,-0.0400,1.0000
C00645=-119.950,31.510,70.770,-0.0400,-0.0000,1.0000
C00646=-119.010,37.980,71.130,-0.0000,0.0000,1.0000
C00647=-116.780,44.550,71.370,-0.0000,0.0000,1.0000
C00648=-114.080,51.070,71.370,-0.0000,0.0000,1.0000
C00649=-111.010,57.300,71.130,-0.0000,0.0000,1.0000
C00650=-107.100,62.540,70.770,-0.0300,0.0300,1.0000
C00651=-101.780,65.420,70.410,-0.0200,0.0800,1.0000
C00652=-96.130,65.450,69.980,0.0400,0.1300,0.9900
C00653=-90.930,62.780,69.160,0.0600,0.1200,0.9900
C00654=-85.680,59.550,67.530,0.0500,0.0800,1.0000
C00655=-80.980,56.760,65.440,0.0100,0.0200,1.0000
C00656=-77.140,55.080,63.440,-0.0400,-0.1200,0.9900
C00657=-73.860,55.310,62.020,0.1800,-0.5000,0.8400
C00658=-70.380,58.280,61.450,0.4400,-0.4400,0.7800
C00659=-67.450,61.560,61.430,0.4700,-0.4200,0.7700
C00660=-64.570,64.570,61.440,0.4500,-0.4500,0.7700
C00661=-61.560,67.450,61.430,0.4200,-0.4700,0.7700
C00662=-58.280,70.380,61.450,0.4400,-0.4400,0.7800
C00663=-55.310,73.860,62.020,0.5000,-0.1800,0.8400
C00664=-55.080,77.140,63.440,0.1200,0.0400,0.9900
C00665=-56.760,80.980,65.440,-0.0200,-0.0100,1.0000
C00666=-59.550,85.680,67.530,-0.0800,-0.0500,1.0000
C00667=-62.780,90.930,69.160,-0.1200,-0.0600,0.9900
C00668=-65.450,96.130,69.980,-0.1300,-0.0400,0.9900
C00669=-65.420,101.780,70.410,-0.0800,0.0200,1.0000
C00670=-62.540,107.100,70.770,-0.0300,0.0300,1.0000
C00671=-57.300,111.010,71.130,-0.0000,0.0000,1.0000
C00672=-51.070,114.080,71.370,-0.0000,0.0000,1.0000
C00673=-44.550,116.780,71.370,-0.0000,0.0000,1.0000
C00674=-37.980,119.010,71.130,-0.0000,0.0000,1.0000
C00675=-31.510,119.950,70.770,0.0000,0.0400,1.0000
C00676=-25.720,118.230,70.410,0.0400,0.0700,1.0000
C00677=-21.690,114.260,69.980,0.1200,0.0700,0.9900
C00678=-19.900,108.690,69.160,0.1300,0.0400,0.9900
C00679=-18.480,102.690,67.530,0.0900,0.0200,1.0000
C00680=-17.130,97.400,65.440,0.0200,0.0100,1.0000
C00681=-15.600,93.500,63.440,-0.1100,-0.0500,0.9900
C00682=-13.120,91.330,62.020,-0.2300,-0.4900,0.8400
C00683=-8.560,90.970,61.450,0.0000,-0.6300,0.7800
C00684=-4.160,91.220,61.430,0.0300,-0.6300,0.7700
C00685=0.000,91.320,61.440,-0.0000,-0.6300,0.7700
C00686=0.000,90.240,62.760,-0.0000,-0.6300,0.7700
C00687=-4.060,90.150,62.740,0.0300,-0.6300,0.7700
C00688=-8.390,89.910,62.770,-0.0000,-0.6300,0.7800
C00689=-12.910,90.310,63.350,-0.2300,-0.4700,0.8500
C00690=-15.350,92.560,64.840,-0.1000,-0.0500,0.9900
C00691=-16.840,96.600,66.910,0.0300,0.0100,1.0000
C00692=-18.160,102.080,69.090,0.0900,0.0200,1.0000
C00693=-19.560,108.290,70.780,0.1300,0.0400,0.9900
C00694=-21.320,114.060,71.630,0.1200,0.0600,0.9900
C00695=-25.370,118.190,72.080,0.0400,0.0700,1.0000
C00696=-31.240,120.000,72.450,0.0000,0.0400,1.0000
C00697=-37.800,119.070,72.820,-0.0000,0.0000,1.0000
C00698=-44.490,116.800,73.070,-0.0000,0.0000,1.0000
C00699=-51.130,114.050,73.070,-0.0000,0.0000,1.0000
C00700=-57.460,110.930,72.820,-0.0000,0.0000,1.0000
C00701=-62.770,106.940,72.450,-0.0300,0.0300,1.0000
C00702=-65.630,101.510,72.080,-0.0800,0.0200,1.0000
C00703=-65.570,95.730,71.630,-0.1300,-0.0400,0.9900
C00704=-62.740,90.410,70.780,-0.1200,-0.0700,0.9900
C00705=-59.330,85.020,69.090,-0.0800,-0.0500,1.0000
C00706=-56.400,80.210,66.910,-0.0300,-0.0200,1.0000
C00707=-54.590,76.300,64.840,0.1100,0.0400,0.9900
C00708=-54.720,72.990,63.350,0.5000,-0.1700,0.8500
C00709=-57.640,69.510,62.770,0.4500,-0.4400,0.7800
C00710=-60.870,66.620,62.740,0.4200,-0.4700,0.7700
C00711=-63.810,63.810,62.760,0.4500,-0.4500,0.7700
C00712=-66.620,60.870,62.740,0.4700,-0.4200,0.7700
C00713=-69.510,57.640,62.770,0.4400,-0.4500,0.7800
C00714=-72.990,54.720,63.350,0.1700,-0.5000,0.8500
C00715=-76.300,54.590,64.840,-0.0400,-0.1100,0.9900
C00716=-80.210,56.400,66.910,0.0200,0.0300,1.0000
C00717=-85.020,59.330,69.090,0.0500,0.0800,1.0000
C00718=-90.410,62.740,70.780,0.0700,0.1200,0.9900
C00719=-95.730,65.570,71.630,0.0400,0.1300,0.9900
C00720=-101.510,65.630,72.080,-0.0200,0.0800,1.0000
C00721=-106.940,62.770,72.450,-0.0300,0.0300,1.0000
C00722=-110.930,57.460,72.820,-0.0000,0.0000,1.0000
C00723=-114.050,51.130,73.070,-0.0000,0.0000,1.0000
C00724=-116.800,44.490,73.070,-0.0000,0.0000,1.0000
C00725=-119.070,37.800,72.820,-0.0000,0.0000,1.0000
C00726=-120.000,31.240,72.450,-0.0400,-0.0000,1.0000
C00727=-118.190,25.370,72.080,-0.0700,-0.0400,1.0000
C00728=-114.060,21.320,71.630,-0.0600,-0.1200,0.9900
C00729=-108.290,19.560,70.780,-0.0400,-0.1300,0.9900
C00730=-102.080,18.160,69.090,-0.0200,-0.0900,1.0000
C00731=-96.600,16.840,66.910,-0.0100,-0.0300,1.0000
C00732=-92.560,15.350,64.840,0.0500,0.1000,0.9900
C00733=-90.310,12.910,63.350,0.4700,0.2300,0.8500
C00734=-89.910,8.390,62.770,0.6300,0.0000,0.7800
C00735=-90.150,4.060,62.740,0.6300,-0.0300,0.7700
C00736=-90.240,0.000,62.760,0.6300,0.0000,0.7700
C00737=-90.150,-4.060,62.740,0.6300,0.0300,0.7700
C00738=-89.910,-8.390,62.770,0.6300,-0.0000,0.7800
C00739=-90.310,-12.910,63.350,0.4700,-0.2300,0.8500
C00740=-92.560,-15.350,64.840,0.0500,-0.1000,0.9900
C00741=-96.600,-16.840,66.910,-0.0100,0.0300,1.0000
C00742=-102.080,-18.160,69.090,-0.0200,0.0900,1.0000
C00743=-108.290,-19.560,70.780,-0.0400,0.1300,0.9900
C00744=-114.060,-21.320,71.630,-0.0600,0.1200,0.9900
C00745=-118.190,-25.370,72.080,-0.0700,0.0400,1.0000
C00746=-120.000,-31.240,72.450,-0.0400,0.0000,1.0000
C00747=-119.070,-37.800,72.820,-0.0000,-0.0000,1.0000
C00748=-116.800,-44.490,73.070,-0.0000,-0.0000,1.0000
C00749=-114.050,-51.130,73.070,-0.0000,-0.0000,1.0000
C00750=-110.930,-57.460,72.820,-0.0000,-0.0000,1.0000
C00751=-106.940,-62.770,72.450,-0.0300,-0.0300,1.0000
C00752=-101.510,-65.630,72.080,-0.0200,-0.0800,1.0000
C00753=-95.730,-65.570,71.630,0.0400,-0.1300,0.9900
C00754=-90.410,-62.740,70.780,0.0700,-0.1200,0.9900
C00755=-85.020,-59.330,69.090,0.0500,-0.0800,1.0000
C00756=-80.210,-56.400,66.910,0.0200,-0.0300,1.0000
C00757=-76.300,-54.590,64.840,-0.0400,0.1100,0.9900
C00758=-72.990,-54.720,63.350,0.1700,0.5000,0.8500
C00759=-69.510,-57.640,62.770,0.4400,0.4500,0.7800
C00760=-66.620,-60.870,62.740,0.4700,0.4200,0.7700
C00761=-63.810,-63.810,62.760,0.4500,0.4500,0.7700
C00762=-60.870,-66.620,62.740,0.4200,0.4700,0.7700
C00763=-57.640,-69.510,62.770,0.4500,0.4400,0.7800
C00764=-54.720,-72.990,63.350,0.5000,0.1700,0.8500
C00765=-54.590,-76.300,64.840,0.1100,-0.0400,0.9900
C00766=-56.400,-80.210,66.910,-0.0300,0.0200,1.0000
C00767=-59.330,-85.020,69.090,-0.0800,0.0500,1.0000
C00768=-62.740,-90.410,70.780,-0.1200,0.0700,0.9900
C00769=-65.570,-95.730,71.630,-0.1300,0.0400,0.9900
C00770=-65.630,-101.510,72.080,-0.0800,-0.0200,1.0000
C00771=-62.770,-106.940,72.450,-0.0300,-0.0300,1.0000
C00772=-57.460,-110.930,72.820,-0.0000,-0.0000,1.0000
C00773=-51.130,-114.050,73.070,-0.0000,-0.0000,1.0000
C00774=-44.490,-116.800,73.070,-0.0000,-0.0000,1.0000
C00775=-37.800,-119.070,72.820,-0.0000,-0.0000,1.0000
C00776=-31.240,-120.000,72.450,0.0000,-0.0400,1.0000
C00777=-25.370,-118.190,72.080,0.0400,-0.0700,1.0000
C00778=-21.320,-114.060,71.630,0.1200,-0.0600,0.9900
C00779=-19.560,-108.290,70.780,0.1300,-0.0400,0.9900
C00780=-18.160,-102.080,69.090,0.0900,-0.0200,1.0000
C00781=-16.840,-96.600,66.910,0.0300,-0.0100,1.0000
C00782=-15.350,-92.560,64.840,-0.1000,0.0500,0.9900
C00783=-12.910,-90.310,63.350,-0.2300,0.4700,0.8500
C00784=-8.390,-89.910,62.770,-0.0000,0.6300,0.7800
C00785=-4.060,-90.150,62.740,0.0300,0.6300,0.7700
C00786=0.000,-90.240,62.760,-0.0000,0.6300,0.7700
C00787=0.000,-90.240,62.760,-0.0000,0.6300,0.7700
C00788=4.060,-90.150,62.740,-0.0300,0.6300,0.7700
C00789=8.390,-89.910,62.770,0.0000,0.6300,0.7800
C00790=12.910,-90.310,63.350,0.2300,0.4700,0.8500
C00791=15.350,-92.560,64.840,0.1000,0.0500,0.9900
C00792=16.840,-96.600,66.910,-0.0300,-0.0100,1.0000
C00793=18.160,-102.080,69.090,-0.0900,-0.0200,1.0000
C00794=19.560,-108.290,70.780,-0.1300,-0.0400,0.9900
C00795=21.320,-114.060,71.630,-0.1200,-0.0600,0.9900
C00796=25.370,-118.190,72.080,-0.0400,-0.0700,1.0000
C00797=31.240,-120.000,72.450,-0.0000,-0.0400,1.0000
C00798=37.800,-119.070,72.820,0.0000,-0.0000,1.0000
C00799=44.490,-116.800,73.070,0.0000,-0.0000,1.0000
C00800=51.130,-114.050,73.070,0.0000,-0.0000,1.0000
C00801=57.460,-110.930,72.820,0.0000,-0.0000,1.0000
C00802=62.770,-106.940,72.450,0.0300,-0.0300,1.0000
C00803=65.630,-101.510,72.080,0.0800,-0.0200,1.0000
C00804=65.570,-95.730,71.630,0.1300,0.0400,0.9900
C00805=62.740,-90.410,70.780,0.1200,0.0700,0.9900
C00806=59.330,-85.020,69.090,0.0800,0.0500,1.0000
C00807=56.400,-80.210,66.910,0.0300,0.0200,1.0000
C00808=54.590,-76.300,64.840,-0.1100,-0.0400,0.9900
C00809=54.720,-72.990,63.350,-0.5000,0.1700,0.8500
C00810=57.640,-69.510,62.770,-0.4500,0.4400,0.7800
C00811=60.870,-66.620,62.740,-0.4200,0.4700,0.7700
C00812=63.810,-63.810,62.760,-0.4500,0.4500,0.7700
C00813=66.620,-60.870,62.740,-0.4700,0.4200,0.7700
C00814=69.510,-57.640,62.770,-0.4400,0.4500,0.7800
C00815=72.990,-54.720,63.350,-0.1700,0.5000,0.8500
C00816=76.300,-54.590,64.840,0.0400,0.1100,0.9900
C00817=80.210,-56.400,66.910,-0.0200,-0.0300,1.0000
C00818=85.020,-59.330,69.090,-0.0500,-0.0800,1.0000
C00819=90.410,-62.740,70.780,-0.0700,-0.1200,0.9900
C00820=95.730,-65.570,71.630,-0.0400,-0.1300,0.9900
C00821=101.510,-65.630,72.080,0.0200,-0.0800,1.0000
C00822=106.940,-62.770,72.450,0.0300,-0.0300,1.0000
C00823=110.930,-57.460,72.820,0.0000,-0.0000,1.0000
C00824=114.050,-51.130,73.070,0.0000,-0.0000,1.0000
C00825=116.800,-44.490,73.070,0.0000,-0.0000,1.0000
C00826=119.070,-37.800,72.820,0.0000,-0.0000,1.0000
C00827=120.000,-31.240,72.450,0.0400,0.0000,1.0000
C00828=118.190,-25.370,72.080,0.0700,0.0400,1.0000
C00829=114.060,-21.320,71.630,0.0600,0.1200,0.9900
C00830=108.290,-19.560,70.780,0.0400,0.1300,0.9900
C00831=102.080,-18.160,69.090,0.0200,0.0900,1.0000
C00832=96.600,-16.840,66.910,0.0100,0.0300,1.0000
C00833=92.560,-15.350,64.840,-0.0500,-0.1000,0.9900
C00834=90.310,-12.910,63.350,-0.4700,-0.2300,0.8500
C00835=89.910,-8.390,62.770,-0.6300,-0.0000,0.7800
C00836=90.150,-4.060,62.740,-0.6300,0.0300,0.7700
C00837=90.240,0.000,62.760,-0.6300,-0.0000,0.7700
C00838=90.150,4.060,62.740,-0.6300,-0.0300,0.7700
C00839=89.910,8.390,62.770,-0.6300,0.0000,0.7800
C00840=90.310,12.910,63.350,-0.4700,0.2300,0.8500
C00841=92.560,15.350,64.840,-0.0500,0.1000,0.9900
C00842=96.600,16.840,66.910,0.0100,-0.0300,1.0000
C00843=102.080,18.160,69.090,0.0200,-0.0900,1.0000
C00844=108.290,19.560,70.780,0.0400,-0.1300,0.9900
C00845=114.060,21.320,71.630,0.0600,-0.1200,0.9900
C00846=118.190,25.370,72.080,0.0700,-0.0400,1.0000
C00847=120.000,31.240,72.450,0.0400,-0.0000,1.0000
C00848=119.070,37.800,72.820,0.0000,0.0000,1.0000
C00849=116.800,44.490,73.070,0.0000,0.0000,1.0000
C00850=114.050,51.130,73.070,0.0000,0.0000,1.0000
C00851=110.930,57.460,72.820,0.0000,0.0000,1.0000
C00852=106.940,62.770,72.450,0.0300,0.0300,1.0000
C00853=101.510,65.630,72.080,0.0200,0.0800,1.0000
C00854=95.730,65.570,71.630,-0.0400,0.1300,0.9900
C00855=90.410,62.740,70.780,-0.0700,0.1200,0.9900
C00856=85.020,59.330,69.090,-0.0500,0.0800,1.0000
C00857=80.210,56.400,66.910,-0.0200,0.0300,1.0000
C00858=76.300,54.590,64.840,0.0400,-0.1100,0.9900
C00859=72.990,54.720,63.350,-0.1700,-0.5000,0.8500
C00860=69.510,57.640,62.770,-0.4400,-0.4500,0.7800
C00861=66.620,60.870,62.740,-0.4700,-0.4200,0.7700
C00862=63.810,63.810,62.760,-0.4500,-0.4500,0.7700
C00863=60.870,66.620,62.740,-0.4200,-0.4700,0.7700
C00864=57.640,69.510,62.770,-0.4500,-0.4400,0.7800
C00865=54.720,72.990,63.350,-0.5000,-0.1700,0.8500
C00866=54.590,76.300,64.840,-0.1100,0.0400,0.9900
C00867=56.400,80.210,66.910,0.0300,-0.0200,1.0000
C00868=59.330,85.020,69.090,0.0800,-0.0500,1.0000
C00869=62.740,90.410,70.780,0.1200,-0.0700,0.9900
C00870=65.570,95.730,71.630,0.1300,-0.0400,0.9900
C00871=65.630,101.510,72.080,0.0800,0.0200,1.0000
C00872=62.770,106.940,72.450,0.0300,0.0300,1.0000
C00873=57.460,110.930,72.820,0.0000,0.0000,1.0000
C00874=51.130,114.050,73.070,0.0000,0.0000,1.0000
C00875=44.490,116.800,73.070,0.0000,0.0000,1.0000
C00876=37.800,119.070,72.820,0.0000,0.0000,1.0000
C00877=31.240,120.000,72.450,-0.0000,0.0400,1.0000
C00878=25.370,118.190,72.080,-0.0400,0.0700,1.0000
C00879=21.320,114.060,71.630,-0.1200,0.0600,0.9900
C00880=19.560,108.290,70.780,-0.1300,0.0400,0.9900
C00881=18.160,102.080,69.090,-0.0900,0.0200,1.0000
C00882=16.840,96.600,66.910,-0.0300,0.0100,1.0000
C00883=15.350,92.560,64.840,0.1000,-0.0500,0.9900
C00884=12.910,90.310,63.350,0.2300,-0.4700,0.8500
C00885=8.390,89.910,62.770,0.0000,-0.6300,0.7800
C00886=4.060,90.150,62.740,-0.0300,-0.6300,0.7700
C00887=0.000,90.240,62.760,-0.0000,-0.6300,0.7700
C00888=0.000,89.170,64.080,-0.0000,-0.6300,0.7800
C00889=3.970,89.080,64.060,-0.0300,-0.6300,0.7800
C00890=8.230,88.850,64.090,0.0100,-0.6300,0.7800
C00891=12.710,89.280,64.690,0.2400,-0.4600,0.8500
C00892=15.100,91.620,66.230,0.0900,-0.0400,1.0000
C00893=16.560,95.800,68.390,-0.0400,0.0100,1.0000
C00894=17.850,101.470,70.640,-0.1000,0.0200,0.9900
C00895=19.230,107.890,72.400,-0.1300,0.0300,0.9900
C00896=20.960,113.860,73.280,-0.1200,0.0600,0.9900
C00897=25.030,118.150,73.740,-0.0400,0.0700,1.0000
C00898=30.970,120.050,74.120,-0.0000,0.0400,1.0000
C00899=37.630,119.130,74.510,0.0000,0.0000,1.0000
C00900=44.430,116.830,74.770,0.0000,0.0000,1.0000
C00901=51.190,114.030,74.770,0.0000,0.0000,1.0000
C00902=57.630,110.840,74.510,0.0000,0.0000,1.0000
C00903=62.990,106.790,74.120,0.0300,0.0300,1.0000
C00904=65.840,101.240,73.740,0.0800,0.0200,1.0000
C00905=65.690,95.330,73.280,0.1300,-0.0400,0.9900
C00906=62.690,89.890,72.400,0.1200,-0.0700,0.9900
C00907=59.120,84.370,70.640,0.0900,-0.0500,0.9900
C00908=56.030,79.450,68.390,0.0300,-0.0200,1.0000
C00909=54.110,75.460,66.230,-0.0900,0.0400,1.0000
C00910=54.140,72.120,64.690,-0.5000,-0.1600,0.8500
C00911=57.010,68.650,64.090,-0.4500,-0.4400,0.7800
C00912=60.190,65.790,64.060,-0.4200,-0.4700,0.7800
C00913=63.050,63.050,64.080,-0.4500,-0.4500,0.7800
C00914=65.790,60.190,64.060,-0.4700,-0.4200,0.7800
C00915=68.650,57.010,64.090,-0.4400,-0.4500,0.7800
C00916=72.120,54.140,64.690,-0.1600,-0.5000,0.8500
C00917=75.460,54.110,66.230,0.0400,-0.0900,1.0000
C00918=79.450,56.030,68.390,-0.0200,0.0300,1.0000
C00919=84.370,59.120,70.640,-0.0500,0.0900,0.9900
C00920=89.890,62.690,72.400,-0.0700,0.1200,0.9900
C00921=95.330,65.690,73.280,-0.0400,0.1300,0.9900
C00922=101.240,65.840,73.740,0.0200,0.0800,1.0000
C00923=106.790,62.990,74.120,0.0300,0.0300,1.0000
C00924=110.840,57.630,74.510,0.0000,0.0000,1.0000
C00925=114.030,51.190,74.770,0.0000,0.0000,1.0000
C00926=116.830,44.430,74.770,0.0000,0.0000,1.0000
C00927=119.130,37.630,74.510,0.0000,0.0000,1.0000
C00928=120.050,30.970,74.120,0.0400,-0.0000,1.0000
C00929=118.150,25.030,73.740,0.0700,-0.0400,1.0000
C00930=113.860,20.960,73.280,0.0600,-0.1200,0.9900
C00931=107.890,19.230,72.400,0.0300,-0.1300,0.9900
C00932=101.470,17.850,70.640,0.0200,-0.1000,0.9900
C00933=95.800,16.560,68.390,0.0100,-0.0400,1.0000
C00934=91.620,15.100,66.230,-0.0400,0.0900,1.0000
C00935=89.280,12.710,64.690,-0.4600,0.2400,0.8500
C00936=88.850,8.230,64.090,-0.6300,0.0100,0.7800
C00937=89.080,3.970,64.060,-0.6300,-0.0300,0.7800
C00938=89.170,0.000,64.080,-0.6300,-0.0000,0.7800
C00939=89.080,-3.970,64.060,-0.6300,0.0300,0.7800
C00940=88.850,-8.230,64.090,-0.6300,-0.0100,0.7800
C00941=89.280,-12.710,64.690,-0.4600,-0.2400,0.8500
C00942=91.620,-15.100,66.230,-0.0400,-0.0900,1.0000
C00943=95.800,-16.560,68.390,0.0100,0.0400,1.0000
C00944=101.470,-17.850,70.640,0.0200,0.1000,0.9900
C00945=107.890,-19.230,72.400,0.0300,0.1300,0.9900
C00946=113.860,-20.960,73.280,0.0600,0.1200,0.9900
C00947=118.150,-25.030,73.740,0.0700,0.0400,1.0000
C00948=120.050,-30.970,74.120,0.0400,0.0000,1.0000
C00949=119.130,-37.630,74.510,0.0000,-0.0000,1.0000
C00950=116.830,-44.430,74.770,0.0000,-0.0000,1.0000
C00951=114.030,-51.190,74.770,0.0000,-0.0000,1.0000
C00952=110.840,-57.630,74.510,0.0000,-0.0000,1.0000
C00953=106.790,-62.990,74.120,0.0300,-0.0300,1.0000
C00954=101.240,-65.840,73.740,0.0200,-0.0800,1.0000
C00955=95.330,-65.690,73.280,-0.0400,-0.1300,0.9900
C00956=89.890,-62.690,72.400,-0.0700,-0.1200,0.9900
C00957=84.370,-59.120,70.640,-0.0500,-0.0900,0.9900
C00958=79.450,-56.030,68.390,-0.0200,-0.0300,1.0000
C00959=75.460,-54.110,66.230,0.0400,0.0900,1.0000
C00960=72.120,-54.140,64.690,-0.1600,0.5000,0.8500
C00961=68.650,-57.010,64.090,-0.4400,0.4500,0.7800
C00962=65.790,-60.190,64.060,-0.4700,0.4200,0.7800
C00963=63.050,-63.050,64.080,-0.4500,0.4500,0.7800
C00964=60.190,-65.790,64.060,-0.4200,0.4700,0.7800
C00965=57.010,-68.650,64.090,-0.4500,0.4400,0.7800
C00966=54.140,-72.120,64.690,-0.5000,0.1600,0.8500
C00967=54.110,-75.460,66.230,-0.0900,-0.0400,1.0000
C00968=56.030,-79.450,68.390,0.0300,0.0200,1.0000
C00969=59.120,-84.370,70.640,0.0900,0.0500,0.9900
C00970=62.690,-89.890,72.400,0.1200,0.0700,0.9900
C00971=65.690,-95.330,73.280,0.1300,0.0400,0.9900
C00972=65.840,-101.240,73.740,0.0800,-0.0200,1.0000
C00973=62.990,-106.790,74.120,0.0300,-0.0300,1.0000
C00974=57.630,-110.840,74.510,0.0000,-0.0000,1.0000
C00975=51.190,-114.030,74.770,0.0000,-0.0000,1.0000
C00976=44.430,-116.830,74.770,0.0000,-0.0000,1.0000
C00977=37.630,-119.130,74.510,0.0000,-0.0000,1.0000
C00978=30.970,-120.050,74.120,-0.0000,-0.0400,1.0000
C00979=25.030,-118.150,73.740,-0.0400,-0.0700,1.0000
C00980=20.960,-113.860,73.280,-0.1200,-0.0600,0.9900
C00981=19.230,-107.890,72.400,-0.1300,-0.0300,0.9900
C00982=17.850,-101.470,70.640,-0.1000,-0.0200,0.9900
C00983=16.560,-95.800,68.390,-0.0400,-0.0100,1.0000
C00984=15.100,-91.620,66.230,0.0900,0.0400,1.0000
C00985=12.710,-89.280,64.690,0.2400,0.4600,0.8500
C00986=8.230,-88.850,64.090,0.0100,0.6300,0.7800
C00987=3.970,-89.080,64.060,-0.0300,0.6300,0.7800
C00988=0.000,-89.170,64.080,-0.0000,0.6300,0.7800
C00989=0.000,-89.170,64.080,-0.0000,0.6300,0.7800
C00990=-3.970,-89.080,64.060,0.0300,0.6300,0.7800
C00991=-8.230,-88.850,64.090,-0.0100,0.6300,0.7800
C00992=-12.710,-89.280,64.690,-0.2400,0.4600,0.8500
C00993=-15.100,-91.620,66.230,-0.0900,0.0400,1.0000
C00994=-16.560,-95.800,68.390,0.0400,-0.0100,1.0000
C00995=-17.850,-101.470,70.640,0.1000,-0.0200,0.9900
C00996=-19.230,-107.890,72.400,0.1300,-0.0300,0.9900
C00997=-20.960,-113.860,73.280,0.1200,-0.0600,0.9900
C00998=-25.030,-118.150,73.740,0.0400,-0.0700,1.0000
C00999=-30.970,-120.050,74.120,0.0000,-0.0400,1.0000
C01000=-37.630,-119.130,74.510,-0.0000,-0.0000,1.0000
C01001=-44.430,-116.830,74.770,-0.0000,-0.0000,1.0000
C01002=-51.190,-114.030,74.770,-0.0000,-0.0000,1.0000
C01003=-57.630,-110.840,74.510,-0.0000,-0.0000,1.0000
C01004=-62.990,-106.790,74.120,-0.0300,-0.0300,1.0000
C01005=-65.840,-101.240,73.740,-0.0800,-0.0200,1.0000
C01006=-65.690,-95.330,73.280,-0.1300,0.0400,0.9900
C01007=-62.690,-89.890,72.400,-0.1200,0.0700,0.9900
C01008=-59.120,-84.370,70.640,-0.0900,0.0500,0.9900
C01009=-56.030,-79.450,68.390,-0.0300,0.0200,1.0000
C01010=-54.110,-75.460,66.230,0.0900,-0.0400,1.0000
C01011=-54.140,-72.120,64.690,0.5000,0.1600,0.8500
C01012=-57.010,-68.650,64.090,0.4500,0.4400,0.7800
C01013=-60.190,-65.790,64.060,0.4200,0.4700,0.7800
C01014=-63.050,-63.050,64.080,0.4500,0.4500,0.7800
C01015=-65.790,-60.190,64.060,0.4700,0.4200,0.7800
C01016=-68.650,-57.010,64.090,0.4400,0.4500,0.7800
C01017=-72.120,-54.140,64.690,0.1600,0.5000,0.8500
C01018=-75.460,-54.110,66.230,-0.0400,0.0900,1.0000
C01019=-79.450,-56.030,68.390,0.0200,-0.0300,1.0000
C01020=-84.370,-59.120,70.640,0.0500,-0.0900,0.9900
C01021=-89.890,-62.690,72.400,0.0700,-0.1200,0.9900
C01022=-95.330,-65.690,73.280,0.0400,-0.1300,0.9900
C01023=-101.240,-65.840,73.740,-0.0200,-0.0800,1.0000
C01024=-106.790,-62.990,74.120,-0.0300,-0.0300,1.0000
C01025=-110.840,-57.630,74.510,-0.0000,-0.0000,1.0000
C01026=-114.030,-51.190,74.770,-0.0000,-0.0000,1.0000
C01027=-116.830,-44.430,74.770,-0.0000,-0.0000,1.0000
C01028=-119.130,-37.630,74.510,-0.0000,-0.0000,1.0000
C01029=-120.050,-30.970,74.120,-0.0400,0.0000,1.0000
C01030=-118.150,-25.030,73.740,-0.0700,0.0400,1.0000
C01031=-113.860,-20.960,73.280,-0.0600,0.1200,0.9900
C01032=-107.890,-19.230,72.400,-0.0300,0.1300,0.9900
C01033=-101.470,-17.850,70.640,-0.0200,0.1000,0.9900
C01034=-95.800,-16.560,68.390,-0.0100,0.0400,1.0000
C01035=-91.620,-15.100,66.230,0.0400,-0.0900,1.0000
C01036=-89.280,-12.710,64.690,0.4600,-0.2400,0.8500
C01037=-88.850,-8.230,64.090,0.6300,-0.0100,0.7800
C01038=-89.080,-3.970,64.060,0.6300,0.0300,0.7800
C01039=-89.170,0.000,64.080,0.6300,0.0000,0.7800
C01040=-89.080,3.970,64.060,0.6300,-0.0300,0.7800
C01041=-88.850,8.230,64.090,0.6300,0.0100,0.7800
C01042=-89.280,12.710,64.690,0.4600,0.2400,0.8500
C01043=-91.620,15.100,66.230,0.0400,0.0900,1.0000
C01044=-95.800,16.560,68.390,-0.0100,-0.0400,1.0000
C01045=-101.470,17.850,70.640,-0.0200,-0.1000,0.9900
C01046=-107.890,19.230,72.400,-0.0300,-0.1300,0.9900
C01047=-113.860,20.960,73.280,-0.0600,-0.1200,0.9900
C01048=-118.150,25.030,73.740,-0.0700,-0.0400,1.0000
C01049=-120.050,30.970,74.120,-0.0400,-0.0000,1.0000
C01050=-119.130,37.630,74.510,-0.0000,0.0000,1.0000
C01051=-116.830,44.430,74.770,-0.0000,0.0000,1.0000
C01052=-114.030,51.190,74.770,-0.0000,0.0000,1.0000
C01053=-110.840,57.630,74.510,-0.0000,0.0000,1.0000
C01054=-106.790,62.990,74.120,-0.0300,0.0300,1.0000
C01055=-101.240,65.840,73.740,-0.0200,0.0800,1.0000
C01056=-95.330,65.690,73.280,0.0400,0.1300,0.9900
C01057=-89.890,62.690,72.400,0.0700,0.1200,0.9900
C01058=-84.370,59.120,70.640,0.0500,0.0900,0.9900
C01059=-79.450,56.030,68.390,0.0200,0.0300,1.0000
C01060=-75.460,54.110,66.230,-0.0400,-0.0900,1.0000
C01061=-72.120,54.140,64.690,0.1600,-0.5000,0.8500
C01062=-68.650,57.010,64.090,0.4400,-0.4500,0.7800
C01063=-65.790,60.190,64.060,0.4700,-0.4200,0.7800
C01064=-63.050,63.050,64.080,0.4500,-0.4500,0.7800
C01065=-60.190,65.790,64.060,0.4200,-0.4700,0.7800
C01066=-57.010,68.650,64.090,0.4500,-0.4400,0.7800
C01067=-54.140,72.120,64.690,0.5000,-0.1600,0.8500
C01068=-54.110,75.460,66.230,0.0900,0.0400,1.0000
C01069=-56.030,79.450,68.390,-0.0300,-0.0200,1.0000
C01070=-59.120,84.370,70.640,-0.0900,-0.0500,0.9900
C01071=-62.690,89.890,72.400,-0.1200,-0.0700,0.9900
C01072=-65.690,95.330,73.280,-0.1300,-0.0400,0.9900
C01073=-65.840,101.240,73.740,-0.0800,0.0200,1.0000
C01074=-62.990,106.790,74.120,-0.0300,0.0300,1.0000
C01075=-57.630,110.840,74.510,-0.0000,0.0000,1.0000
C01076=-51.190,114.030,74.770,-0.0000,0.0000,1.0000
C01077=-44.430,116.830,74.770,-0.0000,0.0000,1.0000
C01078=-37.630,119.130,74.510,-0.0000,0.0000,1.0000
C01079=-30.970,120.050,74.120,0.0000,0.0400,1.0000
C01080=-25.030,118.150,73.740,0.0400,0.0700,1.0000
C01081=-20.960,113.860,73.280,0.1200,0.0600,0.9900
C01082=-19.230,107.890,72.400,0.1300,0.0300,0.9900
C01083=-17.850,101.470,70.640,0.1000,0.0200,0.9900
C01084=-16.560,95.800,68.390,0.0400,0.0100,1.0000
C01085=-15.100,91.620,66.230,-0.0900,-0.0400,1.0000
C01086=-12.710,89.280,64.690,-0.2400,-0.4600,0.8500
C01087=-8.230,88.850,64.090,-0.0100,-0.6300,0.7800
C01088=-3.970,89.080,64.060,0.0300,-0.6300,0.7800
C01089=0.000,89.170,64.080,-0.0000,-0.6300,0.7800
C01090=0.000,88.100,65.400,-0.0000,-0.6300,0.7800
C01091=-3.870,88.010,65.380,0.0300,-0.6300,0.7800
C01092=-8.060,87.790,65.410,-0.0100,-0.6200,0.7800
C01093=-12.510,88.250,66.040,-0.2400,-0.4500,0.8600
C01094=-14.850,90.680,67.630,-0.0800,-0.0300,1.0000
C01095=-16.270,95.010,69.860,0.0400,0.0100,1.0000
C01096=-17.540,100.860,72.200,0.1000,0.0200,0.9900
C01097=-18.900,107.500,74.020,0.1300,0.0300,0.9900
C01098=-20.600,113.660,74.930,0.1200,0.0600,0.9900
C01099=-24.690,118.100,75.410,0.0400,0.0700,1.0000
C01100=-30.700,120.100,75.800,0.0000,0.0400,1.0000
C01101=-37.460,119.180,76.200,-0.0000,0.0000,1.0000
C01102=-44.380,116.850,76.460,-0.0000,0.0000,1.0000
C01103=-51.250,114.000,76.460,-0.0000,0.0000,1.0000
C01104=-57.780,110.760,76.200,-0.0000,0.0000,1.0000
C01105=-63.220,106.630,75.800,-0.0300,0.0300,1.0000
C01106=-66.050,100.970,75.410,-0.0800,0.0200,1.0000
C01107=-65.800,94.940,74.930,-0.1300,-0.0400,0.9900
C01108=-62.650,89.370,74.020,-0.1200,-0.0700,0.9900
C01109=-58.920,83.730,72.200,-0.0900,-0.0500,0.9900
C01110=-55.680,78.690,69.860,-0.0400,-0.0200,1.0000
C01111=-53.620,74.630,67.630,0.0800,0.0300,1.0000
C01112=-53.560,71.250,66.040,0.4900,-0.1500,0.8600
C01113=-56.380,67.780,65.410,0.4500,-0.4400,0.7800
C01114=-59.500,64.970,65.380,0.4200,-0.4700,0.7800
C01115=-62.290,62.290,65.400,0.4500,-0.4500,0.7800
C01116=-64.970,59.500,65.380,0.4700,-0.4200,0.7800
C01117=-67.780,56.380,65.410,0.4400,-0.4500,0.7800
C01118=-71.250,53.560,66.040,0.1500,-0.4900,0.8600
C01119=-74.630,53.620,67.630,-0.0300,-0.0800,1.0000
C01120=-78.690,55.680,69.860,0.0200,0.0400,1.0000
C01121=-83.730,58.920,72.200,0.0500,0.0900,0.9900
C01122=-89.370,62.650,74.020,0.0700,0.1200,0.9900
C01123=-94.940,65.800,74.930,0.0400,0.1300,0.9900
C01124=-100.970,66.050,75.410,-0.0200,0.0800,1.0000
C01125=-106.630,63.220,75.800,-0.0300,0.0300,1.0000
C01126=-110.760,57.780,76.200,-0.0000,0.0000,1.0000
C01127=-114.000,51.250,76.460,-0.0000,0.0000,1.0000
C01128=-116.850,44.380,76.460,-0.0000,0.0000,1.0000
C01129=-119.180,37.460,76.200,-0.0000,0.0000,1.0000
C01130=-120.100,30.700,75.800,-0.0400,-0.0000,1.0000
C01131=-118.100,24.690,75.410,-0.0700,-0.0400,1.0000
C01132=-113.660,20.600,74.930,-0.0600,-0.1200,0.9900
C01133=-107.500,18.900,74.020,-0.0300,-0.1300,0.9900
C01134=-100.860,17.540,72.200,-0.0200,-0.1000,0.9900
C01135=-95.010,16.270,69.860,-0.0100,-0.0400,1.0000
C01136=-90.680,14.850,67.630,0.0300,0.0800,1.0000
C01137=-88.250,12.510,66.040,0.4500,0.2400,0.8600
C01138=-87.790,8.060,65.410,0.6200,0.0100,0.7800
C01139=-88.010,3.870,65.380,0.6300,-0.0300,0.7800
C01140=-88.100,0.000,65.400,0.6300,0.0000,0.7800
C01141=-88.010,-3.870,65.380,0.6300,0.0300,0.7800
C01142=-87.790,-8.060,65.410,0.6200,-0.0100,0.7800
C01143=-88.250,-12.510,66.040,0.4500,-0.2400,0.8600
C01144=-90.680,-14.850,67.630,0.0300,-0.0800,1.0000
C01145=-95.010,-16.270,69.860,-0.0100,0.0400,1.0000
C01146=-100.860,-17.540,72.200,-0.0200,0.1000,0.9900
C01147=-107.500,-18.900,74.020,-0.0300,0.1300,0.9900
C01148=-113.660,-20.600,74.930,-0.0600,0.1200,0.9900
C01149=-118.100,-24.690,75.410,-0.0700,0.0400,1.0000
C01150=-120.100,-30.700,75.800,-0.0400,0.0000,1.0000
C01151=-119.180,-37.460,76.200,-0.0000,-0.0000,1.0000
C01152=-116.850,-44.380,76.460,-0.0000,-0.0000,1.0000
C01153=-114.000,-51.250,76.460,-0.0000,-0.0000,1.0000
C01154=-110.760,-57.780,76.200,-0.0000,-0.0000,1.0000
C01155=-106.630,-63.220,75.800,-0.0300,-0.0300,1.0000
C01156=-100.970,-66.050,75.410,-0.0200,-0.0800,1.0000
C01157=-94.940,-65.800,74.930,0.0400,-0.1300,0.9900
C01158=-89.370,-62.650,74.020,0.0700,-0.1200,0.9900
C01159=-83.730,-58.920,72.200,0.0500,-0.0900,0.9900
C01160=-78.690,-55.680,69.860,0.0200,-0.0400,1.0000
C01161=-74.630,-53.620,67.630,-0.0300,0.0800,1.0000
C01162=-71.250,-53.560,66.040,0.1500,0.4900,0.8600
C01163=-67.780,-56.380,65.410,0.4400,0.4500,0.7800
C01164=-64.970,-59.500,65.380,0.4700,0.4200,0.7800
C01165=-62.290,-62.290,65.400,0.4500,0.4500,0.7800
C01166=-59.500,-64.970,65.380,0.4200,0.4700,0.7800
C01167=-56.380,-67.780,65.410,0.4500,0.4400,0.7800
C01168=-53.560,-71.250,66.040,0.4900,0.1500,0.8600
C01169=-53.620,-74.630,67.630,0.0800,-0.0300,1.0000
C01170=-55.680,-78.690,69.860,-0.0400,0.0200,1.0000
C01171=-58.920,-83.730,72.200,-0.0900,0.0500,0.9900
C01172=-62.650,-89.370,74.020,-0.1200,0.0700,0.9900
C01173=-65.800,-94.940,74.930,-0.1300,0.0400,0.9900
C01174=-66.050,-100.970,75.410,-0.0800,-0.0200,1.0000
C01175=-63.220,-106.630,75.800,-0.0300,-0.0300,1.0000
C01176=-57.780,-110.760,76.200,-0.0000,-0.0000,1.0000
C01177=-51.250,-114.000,76.460,-0.0000,-0.0000,1.0000
C01178=-44.380,-116.850,76.460,-0.0000,-0.0000,1.0000
C01179=-37.460,-119.180,76.200,-0.0000,-0.0000,1.0000
C01180=-30.700,-120.100,75.800,0.0000,-0.0400,1.0000
C01181=-24.690,-118.100,75.410,0.0400,-0.0700,1.0000
C01182=-20.600,-113.660,74.930,0.1200,-0.0600,0.9900
C01183=-18.900,-107.500,74.020,0.1300,-0.0300,0.9900
C01184=-17.540,-100.860,72.200,0.1000,-0.0200,0.9900
C01185=-16.270,-95.010,69.860,0.0400,-0.0100,1.0000
C01186=-14.850,-90.680,67.630,-0.0800,0.0300,1.0000
C01187=-12.510,-88.250,66.040,-0.2400,0.4500,0.8600
C01188=-8.060,-87.790,65.410,-0.0100,0.6200,0.7800
C01189=-3.870,-88.010,65.380,0.0300,0.6300,0.7800
C01190=0.000,-88.100,65.400,-0.0000,0.6300,0.7800
C01191=0.000,-88.100,65.400,-0.0000,0.6300,0.7800
C01192=3.870,-88.010,65.380,-0.0300,0.6300,0.7800
C01193=8.060,-87.790,65.410,0.0100,0.6200,0.7800
C01194=12.510,-88.250,66.040,0.2400,0.4500,0.8600
C01195=14.850,-90.680,67.630,0.0800,0.0300,1.0000
C01196=16.270,-95.010,69.860,-0.0400,-0.0100,1.0000
C01197=17.540,-100.860,72.200,-0.1000,-0.0200,0.9900
C01198=18.900,-107.500,74.020,-0.1300,-0.0300,0.9900
C01199=20.600,-113.660,74.930,-0.1200,-0.0600,0.9900
C01200=24.690,-118.100,75.410,-0.0400,-0.0700,1.0000
C01201=30.700,-120.100,75.800,-0.0000,-0.0400,1.0000
C01202=37.460,-119.180,76.200,0.0000,-0.0000,1.0000
C01203=44.380,-116.850,76.460,0.0000,-0.0000,1.0000
C01204=51.250,-114.000,76.460,0.0000,-0.0000,1.0000
C01205=57.780,-110.760,76.200,0.0000,-0.0000,1.0000
C01206=63.220,-106.630,75.800,0.0300,-0.0300,1.0000
C01207=66.050,-100.970,75.410,0.0800,-0.0200,1.0000
C01208=65.800,-94.940,74.930,0.1300,0.0400,0.9900
C01209=62.650,-89.370,74.020,0.1200,0.0700,0.9900
C01210=58.920,-83.730,72.200,0.0900,0.0500,0.9900
C01211=55.680,-78.690,69.860,0.0400,0.0200,1.0000
C01212=53.620,-74.630,67.630,-0.0800,-0.0300,1.0000
C01213=53.560,-71.250,66.040,-0.4900,0.1500,0.8600
C01214=56.380,-67.780,65.410,-0.4500,0.4400,0.7800
C01215=59.500,-64.970,65.380,-0.4200,0.4700,0.7800
C01216=62.290,-62.290,65.400,-0.4500,0.4500,0.7800
C01217=64.970,-59.500,65.380,-0.4700,0.4200,0.7800
C01218=67.780,-56.380,65.410,-0.4400,0.4500,0.7800
C01219=71.250,-53.560,66.040,-0.1500,0.4900,0.8600
C01220=74.630,-53.620,67.630,0.0300,0.0800,1.0000
C01221=78.690,-55.680,69.860,-0.0200,-0.0400,1.0000
C01222=83.730,-58.920,72.200,-0.0500,-0.0900,0.9900
C01223=89.370,-62.650,74.020,-0.0700,-0.1200,0.9900
C01224=94.940,-65.800,74.930,-0.0400,-0.1300,0.9900
C01225=100.970,-66.050,75.410,0.0200,-0.0800,1.0000
C01226=106.630,-63.220,75.800,0.0300,-0.0300,1.0000
C01227=110.760,-57.780,76.200,0.0000,-0.0000,1.0000
C01228=114.000,-51.250,76.460,0.0000,-0.0000,1.0000
C01229=116.850,-44.380,76.460,0.0000,-0.0000,1.0000
C01230=119.180,-37.460,76.200,0.0000,-0.0000,1.0000
C01231=120.100,-30.700,75.800,0.0400,0.0000,1.0000
C01232=118.100,-24.690,75.410,0.0700,0.0400,1.0000
C01233=113.660,-20.600,74.930,0.0600,0.1200,0.9900
C01234=107.500,-18.900,74.020,0.0300,0.1300,0.9900
C01235=100.860,-17.540,72.200,0.0200,0.1000,0.9900
C01236=95.010,-16.270,69.860,0.0100,0.0400,1.0000
C01237=90.680,-14.850,67.630,-0.0300,-0.0800,1.0000
C01238=88.250,-12.510,66.040,-0.4500,-0.2400,0.8600
C01239=87.790,-8.060,65.410,-0.6200,-0.0100,0.7800
C01240=88.010,-3.870,65.380,-0.6300,0.0300,0.7800
C01241=88.100,0.000,65.400,-0.6300,-0.0000,0.7800
C01242=88.010,3.870,65.380,-0.6300,-0.0300,0.7800
C01243=87.790,8.060,65.410,-0.6200,0.0100,0.7800
C01244=88.250,12.510,66.040,-0.4500,0.2400,0.8600
C01245=90.680,14.850,67.630,-0.0300,0.0800,1.0000
C01246=95.010,16.270,69.860,0.0100,-0.0400,1.0000
C01247=100.860,17.540,72.200,0.0200,-0.1000,0.9900
C01248=107.500,18.900,74.020,0.0300,-0.1300,0.9900
C01249=113.660,20.600,74.930,0.0600,-0.1200,0.9900
C01250=118.100,24.690,75.410,0.0700,-0.0400,1.0000
C01251=120.100,30.700,75.800,0.0400,-0.0000,1.0000
C01252=119.180,37.460,76.200,0.0000,0.0000,1.0000
C01253=116.850,44.380,76.460,0.0000,0.0000,1.0000
C01254=114.000,51.250,76.460,0.0000,0.0000,1.0000
C01255=110.760,57.780,76.200,0.0000,0.0000,1.0000
C01256=106.630,63.220,75.800,0.0300,0.0300,1.0000
C01257=100.970,66.050,75.410,0.0200,0.0800,1.0000
C01258=94.940,65.800,74.930,-0.0400,0.1300,0.9900
C01259=89.370,62.650,74.020,-0.0700,0.1200,0.9900
C01260=83.730,58.920,72.200,-0.0500,0.0900,0.9900
C01261=78.690,55.680,69.860,-0.0200,0.0400,1.0000
C01262=74.630,53.620,67.630,0.0300,-0.0800,1.0000
C01263=71.250,53.560,66.040,-0.1500,-0.4900,0.8600
C01264=67.780,56.380,65.410,-0.4400,-0.4500,0.7800
C01265=64.970,59.500,65.380,-0.4700,-0.4200,0.7800
C01266=62.290,62.290,65.400,-0.4500,-0.4500,0.7800
C01267=59.500,64.970,65.380,-0.4200,-0.4700,0.7800
C01268=56.380,67.780,65.410,-0.4500,-0.4400,0.7800
C01269=53.560,71.250,66.040,-0.4900,-0.1500,0.8600
C01270=53.620,74.630,67.630,-0.0800,0.0300,1.0000
C01271=55.680,78.690,69.860,0.0400,-0.0200,1.0000
C01272=58.920,83.730,72.200,0.0900,-0.0500,0.9900
C01273=62.650,89.370,74.020,0.1200,-0.0700,0.9900
C01274=65.800,94.940,74.930,0.1300,-0.0400,0.9900
C01275=66.050,100.970,75.410,0.0800,0.0200,1.0000
C01276=63.220,106.630,75.800,0.0300,0.0300,1.0000
C01277=57.780,110.760,76.200,0.0000,0.0000,1.0000
C01278=51.250,114.000,76.460,0.0000,0.0000,1.0000
C01279=44.380,116.850,76.460,0.0000,0.0000,1.0000
C01280=37.460,119.180,76.200,0.0000,0.0000,1.0000
C01281=30.700,120.100,75.800,-0.0000,0.0400,1.0000
C01282=24.690,118.100,75.410,-0.0400,0.0700,1.0000
C01283=20.600,113.660,74.930,-0.1200,0.0600,0.9900
C01284=18.900,107.500,74.020,-0.1300,0.0300,0.9900
C01285=17.540,100.860,72.200,-0.1000,0.0200,0.9900
C01286=16.270,95.010,69.860,-0.0400,0.0100,1.0000
C01287=14.850,90.680,67.630,0.0800,-0.0300,1.0000
C01288=12.510,88.250,66.040,0.2400,-0.4500,0.8600
C01289=8.060,87.790,65.410,0.0100,-0.6200,0.7800
C01290=3.870,88.010,65.380,-0.0300,-0.6300,0.7800
C01291=0.000,88.100,65.400,-0.0000,-0.6300,0.7800
C01292=0.000,87.030,66.720,-0.0000,-0.6300,0.7800
C01293=3.770,86.950,66.700,-0.0300,-0.6300,0.7800
C01294=7.900,86.740,66.730,0.0100,-0.6200,0.7800
C01295=12.310,87.230,67.380,0.2500,-0.4400,0.8600
C01296=14.610,89.750,69.030,0.0700,-0.0300,1.0000
C01297=15.990,94.220,71.340,-0.0500,0.0100,1.0000
C01298=17.240,100.270,73.760,-0.1000,0.0200,0.9900
C01299=18.570,107.110,75.640,-0.1300,0.0300,0.9900
C01300=20.250,113.470,76.580,-0.1300,0.0600,0.9900
C01301=24.360,118.060,77.080,-0.0500,0.0700,1.0000
C01302=30.430,120.150,77.480,-0.0000,0.0400,1.0000
C01303=37.300,119.240,77.890,0.0000,0.0000,1.0000
C01304=44.320,116.870,78.160,0.0000,0.0000,1.0000
C01305=51.300,113.980,78.160,0.0000,0.0000,1.0000
C01306=57.940,110.690,77.890,0.0000,0.0000,1.0000
C01307=63.440,106.480,77.480,0.0300,0.0300,1.0000
C01308=66.260,100.710,77.080,0.0800,0.0200,1.0000
C01309=65.920,94.550,76.580,0.1300,-0.0500,0.9900
C01310=62.600,88.870,75.640,0.1200,-0.0700,0.9900
C01311=58.710,83.090,73.760,0.0900,-0.0600,0.9900
C01312=55.320,77.930,71.340,0.0400,-0.0300,1.0000
C01313=53.140,73.800,69.030,-0.0700,0.0300,1.0000
C01314=52.980,70.390,67.380,-0.4900,-0.1400,0.8600
C01315=55.750,66.920,66.730,-0.4500,-0.4300,0.7800
C01316=58.810,64.150,66.700,-0.4200,-0.4700,0.7800
C01317=61.540,61.540,66.720,-0.4400,-0.4400,0.7800
C01318=64.150,58.810,66.700,-0.4700,-0.4200,0.7800
C01319=66.920,55.750,66.730,-0.4300,-0.4500,0.7800
C01320=70.390,52.980,67.380,-0.1400,-0.4900,0.8600
C01321=73.800,53.140,69.030,0.0300,-0.0700,1.0000
C01322=77.930,55.320,71.340,-0.0300,0.0400,1.0000
C01323=83.090,58.710,73.760,-0.0600,0.0900,0.9900
C01324=88.870,62.600,75.640,-0.0700,0.1200,0.9900
C01325=94.550,65.920,76.580,-0.0500,0.1300,0.9900
C01326=100.710,66.260,77.080,0.0200,0.0800,1.0000
C01327=106.480,63.440,77.480,0.0300,0.0300,1.0000
C01328=110.690,57.940,77.890,0.0000,0.0000,1.0000
C01329=113.980,51.300,78.160,0.0000,0.0000,1.0000
C01330=116.870,44.320,78.160,0.0000,0.0000,1.0000
C01331=119.240,37.300,77.890,0.0000,0.0000,1.0000
C01332=120.150,30.430,77.480,0.0400,-0.0000,1.0000
C01333=118.060,24.360,77.080,0.0700,-0.0500,1.0000
C01334=113.470,20.250,76.580,0.0600,-0.1300,0.9900
C01335=107.110,18.570,75.640,0.0300,-0.1300,0.9900
C01336=100.270,17.240,73.760,0.0200,-0.1000,0.9900
C01337=94.220,15.990,71.340,0.0100,-0.0500,1.0000
C01338=89.750,14.610,69.030,-0.0300,0.0700,1.0000
C01339=87.230,12.310,67.380,-0.4400,0.2500,0.8600
C01340=86.740,7.900,66.730,-0.6200,0.0100,0.7800
C01341=86.950,3.770,66.700,-0.6300,-0.0300,0.7800
C01342=87.030,0.000,66.720,-0.6300,-0.0000,0.7800
C01343=86.950,-3.770,66.700,-0.6300,0.0300,0.7800
C01344=86.740,-7.900,66.730,-0.6200,-0.0100,0.7800
C01345=87.230,-12.310,67.380,-0.4400,-0.2500,0.8600
C01346=89.750,-14.610,69.030,-0.0300,-0.0700,1.0000
C01347=94.220,-15.990,71.340,0.0100,0.0500,1.0000
C01348=100.270,-17.240,73.760,0.0200,0.1000,0.9900
C01349=107.110,-18.570,75.640,0.0300,0.1300,0.9900
C01350=113.470,-20.250,76.580,0.0600,0.1300,0.9900
C01351=118.060,-24.360,77.080,0.0700,0.0500,1.0000
C01352=120.150,-30.430,77.480,0.0400,0.0000,1.0000
C01353=119.240,-37.300,77.890,0.0000,-0.0000,1.0000
C01354=116.870,-44.320,78.160,0.0000,-0.0000,1.0000
C01355=113.980,-51.300,78.160,0.0000,-0.0000,1.0000
C01356=110.690,-57.940,77.890,0.0000,-0.0000,1.0000
C01357=106.480,-63.440,77.480,0.0300,-0.0300,1.0000
C01358=100.710,-66.260,77.080,0.0200,-0.0800,1.0000
C01359=94.550,-65.920,76.580,-0.0500,-0.1300,0.9900
C01360=88.870,-62.600,75.640,-0.0700,-0.1200,0.9900
C01361=83.090,-58.710,73.760,-0.0600,-0.0900,0.9900
C01362=77.930,-55.320,71.340,-0.0300,-0.0400,1.0000
C01363=73.800,-53.140,69.030,0.0300,0.0700,1.0000
C01364=70.390,-52.980,67.380,-0.1400,0.4900,0.8600
C01365=66.920,-55.750,66.730,-0.4300,0.4500,0.7800
C01366=64.150,-58.810,66.700,-0.4700,0.4200,0.7800
C01367=61.540,-61.540,66.720,-0.4400,0.4400,0.7800
C01368=58.810,-64.150,66.700,-0.4200,0.4700,0.7800
C01369=55.750,-66.920,66.730,-0.4500,0.4300,0.7800
C01370=52.980,-70.390,67.380,-0.4900,0.1400,0.8600
C01371=53.140,-73.800,69.030,-0.0700,-0.0300,1.0000
C01372=55.320,-77.930,71.340,0.0400,0.0300,1.0000
C01373=58.710,-83.090,73.760,0.0900,0.0600,0.9900
C01374=62.600,-88.870,75.640,0.1200,0.0700,0.9900
C01375=65.920,-94.550,76.580,0.1300,0.0500,0.9900
C01376=66.260,-100.710,77.080,0.0800,-0.0200,1.0000
C01377=63.440,-106.480,77.480,0.0300,-0.0300,1.0000
C01378=57.940,-110.690,77.890,0.0000,-0.0000,1.0000
C01379=51.300,-113.980,78.160,0.0000,-0.0000,1.0000
C01380=44.320,-116.870,78.160,0.0000,-0.0000,1.0000
C01381=37.300,-119.240,77.890,0.0000,-0.0000,1.0000
C01382=30.430,-120.150,77.480,-0.0000,-0.0400,1.0000
C01383=24.360,-118.060,77.080,-0.0500,-0.0700,1.0000
C01384=20.250,-113.470,76.580,-0.1300,-0.0600,0.9900
C01385=18.570,-107.110,75.640,-0.1300,-0.0300,0.9900
C01386=17.240,-100.270,73.760,-0.1000,-0.0200,0.9900
C01387=15.990,-94.220,71.340,-0.0500,-0.0100,1.0000
C01388=14.610,-89.750,69.030,0.0700,0.0300,1.0000
C01389=12.310,-87.230,67.380,0.2500,0.4400,0.8600
C01390=7.900,-86.740,66.730,0.0100,0.6200,0.7800
C01391=3.770,-86.950,66.700,-0.0300,0.6300,0.7800
C01392=0.000,-87.030,66.720,-0.0000,0.6300,0.7800
C01393=0.000,-87.030,66.720,-0.0000,0.6300,0.7800
C01394=-3.770,-86.950,66.700,0.0300,0.6300,0.7800
C01395=-7.900,-86.740,66.730,-0.0100,0.6200,0.7800
C01396=-12.310,-87.230,67.380,-0.2500,0.4400,0.8600
C01397=-14.610,-89.750,69.030,-0.0700,0.0300,1.0000
C01398=-15.990,-94.220,71.340,0.0500,-0.0100,1.0000
C01399=-17.240,-100.270,73.760,0.1000,-0.0200,0.9900
C01400=-18.570,-107.110,75.640,0.1300,-0.0300,0.9900
C01401=-20.250,-113.470,76.580,0.1300,-0.0600,0.9900
C01402=-24.360,-118.060,77.080,0.0500,-0.0700,1.0000
C01403=-30.430,-120.150,77.480,0.0000,-0.0400,1.0000
C01404=-37.300,-119.240,77.890,-0.0000,-0.0000,1.0000
C01405=-44.320,-116.870,78.160,-0.0000,-0.0000,1.0000
C01406=-51.300,-113.980,78.160,-0.0000,-0.0000,1.0000
C01407=-57.940,-110.690,77.890,-0.0000,-0.0000,1.0000
C01408=-63.440,-106.480,77.480,-0.0300,-0.0300,1.0000
C01409=-66.260,-100.710,77.080,-0.0800,-0.0200,1.0000
C01410=-65.920,-94.550,76.580,-0.1300,0.0500,0.9900
C01411=-62.600,-88.870,75.640,-0.1200,0.0700,0.9900
C01412=-58.710,-83.090,73.760,-0.0900,0.0600,0.9900
C01413=-55.320,-77.930,71.340,-0.0400,0.0300,1.0000
C01414=-53.140,-73.800,69.030,0.0700,-0.0300,1.0000
C01415=-52.980,-70.390,67.380,0.4900,0.1400,0.8600
C01416=-55.750,-66.920,66.730,0.4500,0.4300,0.7800
C01417=-58.810,-64.150,66.700,0.4200,0.4700,0.7800
C01418=-61.540,-61.540,66.720,0.4400,0.4400,0.7800
C01419=-64.150,-58.810,66.700,0.4700,0.4200,0.7800
C01420=-66.920,-55.750,66.730,0.4300,0.4500,0.7800
C01421=-70.390,-52.980,67.380,0.1400,0.4900,0.8600
C01422=-73.800,-53.140,69.030,-0.0300,0.0700,1.0000
C01423=-77.930,-55.320,71.340,0.0300,-0.0400,1.0000
C01424=-83.090,-58.710,73.760,0.0600,-0.0900,0.9900
C01425=-88.870,-62.600,75.640,0.0700,-0.1200,0.9900
C01426=-94.550,-65.920,76.580,0.0500,-0.1300,0.9900
C01427=-100.710,-66.260,77.080,-0.0200,-0.0800,1.0000
C01428=-106.480,-63.440,77.480,-0.0300,-0.0300,1.0000
C01429=-110.690,-57.940,77.890,-0.0000,-0.0000,1.0000
C01430=-113.980,-51.300,78.160,-0.0000,-0.0000,1.0000
C01431=-116.870,-44.320,78.160,-0.0000,-0.0000,1.0000
C01432=-119.240,-37.300,77.890,-0.0000,-0.0000,1.0000
C01433=-120.150,-30.430,77.480,-0.0400,0.0000,1.0000
C01434=-118.060,-24.360,77.080,-0.0700,0.0500,1.0000
C01435=-113.470,-20.250,76.580,-0.0600,0.1300,0.9900
C01436=-107.110,-18.570,75.640,-0.0300,0.1300,0.9900
C01437=-100.270,-17.240,73.760,-0.0200,0.1000,0.9900
C01438=-94.220,-15.990,71.340,-0.0100,0.0500,1.0000
C01439=-89.750,-14.610,69.030,0.0300,-0.0700,1.0000
C01440=-87.230,-12.310,67.380,0.4400,-0.2500,0.8600
C01441=-86.740,-7.900,66.730,0.6200,-0.0100,0.7800
C01442=-86.950,-3.770,66.700,0.6300,0.0300,0.7800
C01443=-87.030,0.000,66.720,0.6300,0.0000,0.7800
C01444=-86.950,3.770,66.700,0.6300,-0.0300,0.7800
C01445=-86.740,7.900,66.730,0.6200,0.0100,0.7800
C01446=-87.230,12.310,67.380,0.4400,0.2500,0.8600
C01447=-89.750,14.610,69.030,0.0300,0.0700,1.0000
C01448=-94.220,15.990,71.340,-0.0100,-0.0500,1.0000
C01449=-100.270,17.240,73.760,-0.0200,-0.1000,0.9900
C01450=-107.110,18.570,75.640,-0.0300,-0.1300,0.9900
C01451=-113.470,20.250,76.580,-0.0600,-0.1300,0.9900
C01452=-118.060,24.360,77.080,-0.0700,-0.0500,1.0000
C01453=-120.150,30.430,77.480,-0.0400,-0.0000,1.0000
C01454=-119.240,37.300,77.890,-0.0000,0.0000,1.0000
C01455=-116.870,44.320,78.160,-0.0000,0.0000,1.0000
C01456=-113.980,51.300,78.160,-0.0000,0.0000,1.0000
C01457=-110.690,57.940,77.890,-0.0000,0.0000,1.0000
C01458=-106.480,63.440,77.480,-0.0300,0.0300,1.0000
C01459=-100.710,66.260,77.080,-0.0200,0.0800,1.0000
C01460=-94.550,65.920,76.580,0.0500,0.1300,0.9900
C01461=-88.870,62.600,75.640,0.0700,0.1200,0.9900
C01462=-83.090,58.710,73.760,0.0600,0.0900,0.9900
C01463=-77.930,55.320,71.340,0.0300,0.0400,1.0000
C01464=-73.800,53.140,69.030,-0.0300,-0.0700,1.0000
C01465=-70.390,52.980,67.380,0.1400,-0.4900,0.8600
C01466=-66.920,55.750,66.730,0.4300,-0.4500,0.7800
C01467=-64.150,58.810,66.700,0.4700,-0.4200,0.7800
C01468=-61.540,61.540,66.720,0.4400,-0.4400,0.7800
C01469=-58.810,64.150,66.700,0.4200,-0.4700,0.7800
C01470=-55.750,66.920,66.730,0.4500,-0.4300,0.7800
C01471=-52.980,70.390,67.380,0.4900,-0.1400,0.8600
C01472=-53.140,73.800,69.030,0.0700,0.0300,1.0000
C01473=-55.320,77.930,71.340,-0.0400,-0.0300,1.0000
C01474=-58.710,83.090,73.760,-0.0900,-0.0600,0.9900
C01475=-62.600,88.870,75.640,-0.1200,-0.0700,0.9900
C01476=-65.920,94.550,76.580,-0.1300,-0.0500,0.9900
C01477=-66.260,100.710,77.080,-0.0800,0.0200,1.0000
C01478=-63.440,106.480,77.480,-0.0300,0.0300,1.0000
C01479=-57.940,110.690,77.890,-0.0000,0.0000,1.0000
C01480=-51.300,113.980,78.160,-0.0000,0.0000,1.0000
C01481=-44.320,116.870,78.160,-0.0000,0.0000,1.0000
C01482=-37.300,119.240,77.890,-0.0000,0.0000,1.0000
C01483=-30.430,120.150,77.480,0.0000,0.0400,1.0000
C01484=-24.360,118.060,77.080,0.0500,0.0700,1.0000
C01485=-20.250,113.470,76.580,0.1300,0.0600,0.9900
C01486=-18.570,107.110,75.640,0.1300,0.0300,0.9900
C01487=-17.240,100.270,73.760,0.1000,0.0200,0.9900
C01488=-15.990,94.220,71.340,0.0500,0.0100,1.0000
C01489=-14.610,89.750,69.030,-0.0700,-0.0300,1.0000
C01490=-12.310,87.230,67.380,-0.2500,-0.4400,0.8600
C01491=-7.900,86.740,66.730,-0.0100,-0.6200,0.7800
C01492=-3.770,86.950,66.700,0.0300,-0.6300,0.7800
C01493=0.000,87.030,66.720,-0.0000,-0.6300,0.7800
C01494=0.000,85.960,68.040,-0.0000,-0.6300,0.7800
C01495=-3.670,85.880,68.020,0.0300,-0.6300,0.7800
C01496=-7.740,85.680,68.050,-0.0100,-0.6200,0.7800
C01497=-12.110,86.220,68.730,-0.2500,-0.4300,0.8700
C01498=-14.360,88.830,70.440,-0.0600,-0.0200,1.0000
C01499=-15.710,93.440,72.830,0.0500,0.0100,1.0000
C01500=-16.930,99.670,75.330,0.1000,0.0200,0.9900
C01501=-18.250,106.720,77.270,0.1300,0.0300,0.9900
C01502=-19.900,113.280,78.230,0.1300,0.0600,0.9900
C01503=-24.030,118.020,78.740,0.0500,0.0700,1.0000
C01504=-30.180,120.200,79.160,0.0000,0.0400,1.0000
C01505=-37.130,119.290,79.580,-0.0000,0.0000,1.0000
C01506=-44.270,116.890,79.860,-0.0000,0.0000,1.0000
C01507=-51.350,113.960,79.860,-0.0000,0.0000,1.0000
C01508=-58.090,110.610,79.580,-0.0000,0.0000,1.0000
C01509=-63.650,106.330,79.160,-0.0300,0.0300,1.0000
C01510=-66.470,100.450,78.740,-0.0800,0.0200,1.0000
C01511=-66.030,94.170,78.230,-0.1300,-0.0500,0.9900
C01512=-62.560,88.370,77.270,-0.1200,-0.0700,0.9900
C01513=-58.500,82.450,75.330,-0.0900,-0.0600,0.9900
C01514=-54.970,77.180,72.830,-0.0500,-0.0300,1.0000
C01515=-52.660,72.970,70.440,0.0600,0.0300,1.0000
C01516=-52.400,69.520,68.730,0.4800,-0.1200,0.8700
C01517=-55.120,66.060,68.050,0.4500,-0.4300,0.7800
C01518=-58.130,63.330,68.020,0.4200,-0.4600,0.7800
C01519=-60.780,60.780,68.040,0.4400,-0.4400,0.7800
C01520=-63.330,58.130,68.020,0.4600,-0.4200,0.7800
C01521=-66.060,55.120,68.050,0.4300,-0.4500,0.7800
C01522=-69.520,52.400,68.730,0.1200,-0.4800,0.8700
C01523=-72.970,52.660,70.440,-0.0300,-0.0600,1.0000
C01524=-77.180,54.970,72.830,0.0300,0.0500,1.0000
C01525=-82.450,58.500,75.330,0.0600,0.0900,0.9900
C01526=-88.370,62.560,77.270,0.0700,0.1200,0.9900
C01527=-94.170,66.030,78.230,0.0500,0.1300,0.9900
C01528=-100.450,66.470,78.740,-0.0200,0.0800,1.0000
C01529=-106.330,63.650,79.160,-0.0300,0.0300,1.0000
C01530=-110.610,58.090,79.580,-0.0000,0.0000,1.0000
C01531=-113.960,51.350,79.860,-0.0000,0.0000,1.0000
C01532=-116.890,44.270,79.860,-0.0000,0.0000,1.0000
C01533=-119.290,37.130,79.580,-0.0000,0.0000,1.0000
C01534=-120.200,30.180,79.160,-0.0400,-0.0000,1.0000
C01535=-118.020,24.030,78.740,-0.0700,-0.0500,1.0000
C01536=-113.280,19.900,78.230,-0.0600,-0.1300,0.9900
C01537=-106.720,18.250,77.270,-0.0300,-0.1300,0.9900
C01538=-99.670,16.930,75.330,-0.0200,-0.1000,0.9900
C01539=-93.440,15.710,72.830,-0.0100,-0.0500,1.0000
C01540=-88.830,14.360,70.440,0.0200,0.0600,1.0000
C01541=-86.220,12.110,68.730,0.4300,0.2500,0.8700
C01542=-85.680,7.740,68.050,0.6200,0.0100,0.7800
C01543=-85.880,3.670,68.020,0.6300,-0.0300,0.7800
C01544=-85.960,0.000,68.040,0.6300,0.0000,0.7800
C01545=-85.880,-3.670,68.020,0.6300,0.0300,0.7800
C01546=-85.680,-7.740,68.050,0.6200,-0.0100,0.7800
C01547=-86.220,-12.110,68.730,0.4300,-0.2500,0.8700
C01548=-88.830,-14.360,70.440,0.0200,-0.0600,1.0000
C01549=-93.440,-15.710,72.830,-0.0100,0.0500,1.0000
C01550=-99.670,-16.930,75.330,-0.0200,0.1000,0.9900
C01551=-106.720,-18.250,77.270,-0.0300,0.1300,0.9900
C01552=-113.280,-19.900,78.230,-0.0600,0.1300,0.9900
C01553=-118.020,-24.030,78.740,-0.0700,0.0500,1.0000
C01554=-120.200,-30.180,79.160,-0.0400,0.0000,1.0000
C01555=-119.290,-37.130,79.580,-0.0000,-0.0000,1.0000
C01556=-116.890,-44.270,79.860,-0.0000,-0.0000,1.0000
C01557=-113.960,-51.350,79.860,-0.0000,-0.0000,1.0000
C01558=-110.610,-58.090,79.580,-0.0000,-0.0000,1.0000
C01559=-106.330,-63.650,79.160,-0.0300,-0.0300,1.0000
C01560=-100.450,-66.470,78.740,-0.0200,-0.0800,1.0000
C01561=-94.170,-66.030,78.230,0.0500,-0.1300,0.9900
C01562=-88.370,-62.560,77.270,0.0700,-0.1200,0.9900
C01563=-82.450,-58.500,75.330,0.0600,-0.0900,0.9900
C01564=-77.180,-54.970,72.830,0.0300,-0.0500,1.0000
C01565=-72.970,-52.660,70.440,-0.0300,0.0600,1.0000
C01566=-69.520,-52.400,68.730,0.1200,0.4800,0.8700
C01567=-66.060,-55.120,68.050,0.4300,0.4500,0.7800
C01568=-63.330,-58.130,68.020,0.4600,0.4200,0.7800
C01569=-60.780,-60.780,68.040,0.4400,0.4400,0.7800
C01570=-58.130,-63.330,68.020,0.4200,0.4600,0.7800
C01571=-55.120,-66.060,68.050,0.4500,0.4300,0.7800
C01572=-52.400,-69.520,68.730,0.4800,0.1200,0.8700
C01573=-52.660,-72.970,70.440,0.0600,-0.0300,1.0000
C01574=-54.970,-77.180,72.830,-0.0500,0.0300,1.0000
C01575=-58.500,-82.450,75.330,-0.0900,0.0600,0.9900
C01576=-62.560,-88.370,77.270,-0.1200,0.0700,0.9900
C01577=-66.030,-94.170,78.230,-0.1300,0.0500,0.9900
C01578=-66.470,-100.450,78.740,-0.0800,-0.0200,1.0000
C01579=-63.650,-106.330,79.160,-0.0300,-0.0300,1.0000
C01580=-58.090,-110.610,79.580,-0.0000,-0.0000,1.0000
C01581=-51.350,-113.960,79.860,-0.0000,-0.0000,1.0000
C01582=-44.270,-116.890,79.860,-0.0000,-0.0000,1.0000
C01583=-37.130,-119.290,79.580,-0.0000,-0.0000,1.0000
C01584=-30.180,-120.200,79.160,0.0000,-0.0400,1.0000
C01585=-24.030,-118.020,78.740,0.0500,-0.0700,1.0000
C01586=-19.900,-113.280,78.230,0.1300,-0.0600,0.9900
C01587=-18.250,-106.720,77.270,0.1300,-0.0300,0.9900
C01588=-16.930,-99.670,75.330,0.1000,-0.0200,0.9900
C01589=-15.710,-93.440,72.830,0.0500,-0.0100,1.0000
C01590=-14.360,-88.830,70.440,-0.0600,0.0200,1.0000
C01591=-12.110,-86.220,68.730,-0.2500,0.4300,0.8700
C01592=-7.740,-85.680,68.050,-0.0100,0.6200,0.7800
C01593=-3.670,-85.880,68.020,0.0300,0.6300,0.7800
C01594=0.000,-85.960,68.040,-0.0000,0.6300,0.7800
C01595=0.000,-85.960,68.040,-0.0000,0.6300,0.7800
C01596=3.670,-85.880,68.020,-0.0300,0.6300,0.7800
C01597=7.740,-85.680,68.050,0.0100,0.6200,0.7800
C01598=12.110,-86.220,68.730,0.2500,0.4300,0.8700
C01599=14.360,-88.830,70.440,0.0600,0.0200,1.0000
C01600=15.710,-93.440,72.830,-0.0500,-0.0100,1.0000
C01601=16.930,-99.670,75.330,-0.1000,-0.0200,0.9900
C01602=18.250,-106.720,77.270,-0.1300,-0.0300,0.9900
C01603=19.900,-113.280,78.230,-0.1300,-0.0600,0.9900
C01604=24.030,-118.020,78.740,-0.0500,-0.0700,1.0000
C01605=30.180,-120.200,79.160,-0.0000,-0.0400,1.0000
C01606=37.130,-119.290,79.580,0.0000,-0.0000,1.0000
C01607=44.270,-116.890,79.860,0.0000,-0.0000,1.0000
C01608=51.350,-113.960,79.860,0.0000,-0.0000,1.0000
C01609=58.090,-110.610,79.580,0.0000,-0.0000,1.0000
C01610=63.650,-106.330,79.160,0.0300,-0.0300,1.0000
C01611=66.470,-100.450,78.740,0.0800,-0.0200,1.0000
C01612=66.030,-94.170,78.230,0.1300,0.0500,0.9900
C01613=62.560,-88.370,77.270,0.1200,0.0700,0.9900
C01614=58.500,-82.450,75.330,0.0900,0.0600,0.9900
C01615=54.970,-77.180,72.830,0.0500,0.0300,1.0000
C01616=52.660,-72.970,70.440,-0.0600,-0.0300,1.0000
C01617=52.400,-69.520,68.730,-0.4800,0.1200,0.8700
C01618=55.120,-66.060,68.050,-0.4500,0.4300,0.7800
C01619=58.130,-63.330,68.020,-0.4200,0.4600,0.7800
C01620=60.780,-60.780,68.040,-0.4400,0.4400,0.7800
C01621=63.330,-58.130,68.020,-0.4600,0.4200,0.7800
C01622=66.060,-55.120,68.050,-0.4300,0.4500,0.7800
C01623=69.520,-52.400,68.730,-0.1200,0.4800,0.8700
C01624=72.970,-52.660,70.440,0.0300,0.0600,1.0000
C01625=77.180,-54.970,72.830,-0.0300,-0.0500,1.0000
C01626=82.450,-58.500,75.330,-0.0600,-0.0900,0.9900
C01627=88.370,-62.560,77.270,-0.0700,-0.1200,0.9900
C01628=94.170,-66.030,78.230,-0.0500,-0.1300,0.9900
C01629=100.450,-66.470,78.740,0.0200,-0.0800,1.0000
C01630=106.330,-63.650,79.160,0.0300,-0.0300,1.0000
C01631=110.610,-58.090,79.580,0.0000,-0.0000,1.0000
C01632=113.960,-51.350,79.860,0.0000,-0.0000,1.0000
C01633=116.890,-44.270,79.860,0.0000,-0.0000,1.0000
C01634=119.290,-37.130,79.580,0.0000,-0.0000,1.0000
C01635=120.200,-30.180,79.160,0.0400,0.0000,1.0000
C01636=118.020,-24.030,78.740,0.0700,0.0500,1.0000
C01637=113.280,-19.900,78.230,0.0600,0.1300,0.9900
C01638=106.720,-18.250,77.270,0.0300,0.1300,0.9900
C01639=99.670,-16.930,75.330,0.0200,0.1000,0.9900
C01640=93.440,-15.710,72.830,0.0100,0.0500,1.0000
C01641=88.830,-14.360,70.440,-0.0200,-0.0600,1.0000
C01642=86.220,-12.110,68.730,-0.4300,-0.2500,0.8700
C01643=85.680,-7.740,68.050,-0.6200,-0.0100,0.7800
C01644=85.880,-3.670,68.020,-0.6300,0.0300,0.7800
C01645=85.960,0.000,68.040,-0.6300,-0.0000,0.7800
C01646=85.880,3.670,68.020,-0.6300,-0.0300,0.7800
C01647=85.680,7.740,68.050,-0.6200,0.0100,0.7800
C01648=86.220,12.110,68.730,-0.4300,0.2500,0.8700
C01649=88.830,14.360,70.440,-0.0200,0.0600,1.0000
C01650=93.440,15.710,72.830,0.0100,-0.0500,1.0000
C01651=99.670,16.930,75.330,0.0200,-0.1000,0.9900
C01652=106.720,18.250,77.270,0.0300,-0.1300,0.9900
C01653=113.280,19.900,78.230,0.0600,-0.1300,0.9900
C01654=118.020,24.030,78.740,0.0700,-0.0500,1.0000
C01655=120.200,30.180,79.160,0.0400,-0.0000,1.0000
C01656=119.290,37.130,79.580,0.0000,0.0000,1.0000
C01657=116.890,44.270,79.860,0.0000,0.0000,1.0000
C01658=113.960,51.350,79.860,0.0000,0.0000,1.0000
C01659=110.610,58.090,79.580,0.0000,0.0000,1.0000
C01660=106.330,63.650,79.160,0.0300,0.0300,1.0000
C01661=100.450,66.470,78.740,0.0200,0.0800,1.0000
C01662=94.170,66.030,78.230,-0.0500,0.1300,0.9900
C01663=88.370,62.560,77.270,-0.0700,0.1200,0.9900
C01664=82.450,58.500,75.330,-0.0600,0.0900,0.9900
C01665=77.180,54.970,72.830,-0.0300,0.0500,1.0000
C01666=72.970,52.660,70.440,0.0300,-0.0600,1.0000
C01667=69.520,52.400,68.730,-0.1200,-0.4800,0.8700
C01668=66.060,55.120,68.050,-0.4300,-0.4500,0.7800
C01669=63.330,58.130,68.020,-0.4600,-0.4200,0.7800
C01670=60.780,60.780,68.040,-0.4400,-0.4400,0.7800
C01671=58.130,63.330,68.020,-0.4200,-0.4600,0.7800
C01672=55.120,66.060,68.050,-0.4500,-0.4300,0.7800
C01673=52.400,69.520,68.730,-0.4800,-0.1200,0.8700
C01674=52.660,72.970,70.440,-0.0600,0.0300,1.0000
C01675=54.970,77.180,72.830,0.0500,-0.0300,1.0000
C01676=58.500,82.450,75.330,0.0900,-0.0600,0.9900
C01677=62.560,88.370,77.270,0.1200,-0.0700,0.9900
C01678=66.030,94.170,78.230,0.1300,-0.0500,0.9900
C01679=66.470,100.450,78.740,0.0800,0.0200,1.0000
C01680=63.650,106.330,79.160,0.0300,0.0300,1.0000
C01681=58.090,110.610,79.580,0.0000,0.0000,1.0000
C01682=51.350,113.960,79.860,0.0000,0.0000,1.0000
C01683=44.270,116.890,79.860,0.0000,0.0000,1.0000
C01684=37.130,119.290,79.580,0.0000,0.0000,1.0000
C01685=30.180,120.200,79.160,-0.0000,0.0400,1.0000
C01686=24.030,118.020,78.740,-0.0500,0.0700,1.0000
C01687=19.900,113.280,78.230,-0.1300,0.0600,0.9900
C01688=18.250,106.720,77.270,-0.1300,0.0300,0.9900
C01689=16.930,99.670,75.330,-0.1000,0.0200,0.9900
C01690=15.710,93.440,72.830,-0.0500,0.0100,1.0000
C01691=14.360,88.830,70.440,0.0600,-0.0200,1.0000
C01692=12.110,86.220,68.730,0.2500,-0.4300,0.8700
C01693=7.740,85.680,68.050,0.0100,-0.6200,0.7800
C01694=3.670,85.880,68.020,-0.0300,-0.6300,0.7800
C01695=0.000,85.960,68.040,-0.0000,-0.6300,0.7800
C01696=0.000,84.900,69.370,-0.0000,-0.6200,0.7800
C01697=3.580,84.830,69.350,-0.0300,-0.6200,0.7800
C01698=7.570,84.630,69.380,0.0200,-0.6200,0.7900
C01699=11.910,85.200,70.080,0.2600,-0.4200,0.8700
C01700=14.120,87.910,71.850,0.0500,-0.0200,1.0000
C01701=15.430,92.670,74.320,-0.0600,0.0100,1.0000
C01702=16.640,99.090,76.890,-0.1100,0.0200,0.9900
C01703=17.930,106.340,78.890,-0.1300,0.0300,0.9900
C01704=19.550,113.090,79.890,-0.1300,0.0600,0.9900
C01705=23.710,117.990,80.410,-0.0500,0.0700,1.0000
C01706=29.920,120.240,80.840,-0.0000,0.0400,1.0000
C01707=36.970,119.340,81.270,0.0000,0.0000,1.0000
C01708=44.210,116.910,81.560,0.0000,0.0000,1.0000
C01709=51.410,113.930,81.560,0.0000,0.0000,1.0000
C01710=58.240,110.530,81.270,0.0000,0.0000,1.0000
C01711=63.870,106.180,80.840,0.0300,0.0300,1.0000
C01712=66.670,100.190,80.410,0.0800,0.0200,1.0000
C01713=66.140,93.790,79.890,0.1300,-0.0500,0.9900
C01714=62.520,87.880,78.890,0.1200,-0.0700,0.9900
C01715=58.300,81.830,76.890,0.0900,-0.0600,0.9900
C01716=54.620,76.440,74.320,0.0500,-0.0300,1.0000
C01717=52.180,72.140,71.850,-0.0500,0.0200,1.0000
C01718=51.830,68.670,70.080,-0.4700,-0.1100,0.8700
C01719=54.490,65.200,69.380,-0.4500,-0.4200,0.7900
C01720=57.450,62.510,69.350,-0.4200,-0.4600,0.7800
C01721=60.030,60.030,69.370,-0.4400,-0.4400,0.7800
C01722=62.510,57.450,69.350,-0.4600,-0.4200,0.7800
C01723=65.200,54.490,69.380,-0.4200,-0.4500,0.7900
C01724=68.670,51.830,70.080,-0.1100,-0.4700,0.8700
C01725=72.140,52.180,71.850,0.0200,-0.0500,1.0000
C01726=76.440,54.620,74.320,-0.0300,0.0500,1.0000
C01727=81.830,58.300,76.890,-0.0600,0.0900,0.9900
C01728=87.880,62.520,78.890,-0.0700,0.1200,0.9900
C01729=93.790,66.140,79.890,-0.0500,0.1300,0.9900
C01730=100.190,66.670,80.410,0.0200,0.0800,1.0000
C01731=106.180,63.870,80.840,0.0300,0.0300,1.0000
C01732=110.530,58.240,81.270,0.0000,0.0000,1.0000
C01733=113.930,51.410,81.560,0.0000,0.0000,1.0000
C01734=116.910,44.210,81.560,0.0000,0.0000,1.0000
C01735=119.340,36.970,81.270,0.0000,0.0000,1.0000
C01736=120.240,29.920,80.840,0.0400,-0.0000,1.0000
C01737=117.990,23.710,80.410,0.0700,-0.0500,1.0000
C01738=113.090,19.550,79.890,0.0600,-0.1300,0.9900
C01739=106.340,17.930,78.890,0.0300,-0.1300,0.9900
C01740=99.090,16.640,76.890,0.0200,-0.1100,0.9900
C01741=92.670,15.430,74.320,0.0100,-0.0600,1.0000
C01742=87.910,14.120,71.850,-0.0200,0.0500,1.0000
C01743=85.200,11.910,70.080,-0.4200,0.2600,0.8700
C01744=84.630,7.570,69.380,-0.6200,0.0200,0.7900
C01745=84.830,3.580,69.350,-0.6200,-0.0300,0.7800
C01746=84.900,0.000,69.370,-0.6200,-0.0000,0.7800
C01747=84.830,-3.580,69.350,-0.6200,0.0300,0.7800
C01748=84.630,-7.570,69.380,-0.6200,-0.0200,0.7900
C01749=85.200,-11.910,70.080,-0.4200,-0.2600,0.8700
C01750=87.910,-14.120,71.850,-0.0200,-0.0500,1.0000
C01751=92.670,-15.430,74.320,0.0100,0.0600,1.0000
C01752=99.090,-16.640,76.890,0.0200,0.1100,0.9900
C01753=106.340,-17.930,78.890,0.0300,0.1300,0.9900
C01754=113.090,-19.550,79.890,0.0600,0.1300,0.9900
C01755=117.990,-23.710,80.410,0.0700,0.0500,1.0000
C01756=120.240,-29.920,80.840,0.0400,0.0000,1.0000
C01757=119.340,-36.970,81.270,0.0000,-0.0000,1.0000
C01758=116.910,-44.210,81.560,0.0000,-0.0000,1.0000
C01759=113.930,-51.410,81.560,0.0000,-0.0000,1.0000
C01760=110.530,-58.240,81.270,0.0000,-0.0000,1.0000
C01761=106.180,-63.870,80.840,0.0300,-0.0300,1.0000
C01762=100.190,-66.670,80.410,0.0200,-0.0800,1.0000
C01763=93.790,-66.140,79.890,-0.0500,-0.1300,0.9900
C01764=87.880,-62.520,78.890,-0.0700,-0.1200,0.9900
C01765=81.830,-58.300,76.890,-0.0600,-0.0900,0.9900
C01766=76.440,-54.620,74.320,-0.0300,-0.0500,1.0000
C01767=72.140,-52.180,71.850,0.0200,0.0500,1.0000
C01768=68.670,-51.830,70.080,-0.1100,0.4700,0.8700
C01769=65.200,-54.490,69.380,-0.4200,0.4500,0.7900
C01770=62.510,-57.450,69.350,-0.4600,0.4200,0.7800
C01771=60.030,-60.030,69.370,-0.4400,0.4400,0.7800
C01772=57.450,-62.510,69.350,-0.4200,0.4600,0.7800
C01773=54.490,-65.200,69.380,-0.4500,0.4200,0.7900
C01774=51.830,-68.670,70.080,-0.4700,0.1100,0.8700
C01775=52.180,-72.140,71.850,-0.0500,-0.0200,1.0000
C01776=54.620,-76.440,74.320,0.0500,0.0300,1.0000
C01777=58.300,-81.830,76.890,0.0900,0.0600,0.9900
C01778=62.520,-87.880,78.890,0.1200,0.0700,0.9900
C01779=66.140,-93.790,79.890,0.1300,0.0500,0.9900
C01780=66.670,-100.190,80.410,0.0800,-0.0200,1.0000
C01781=63.870,-106.180,80.840,0.0300,-0.0300,1.0000
C01782=58.240,-110.530,81.270,0.0000,-0.0000,1.0000
C01783=51.410,-113.930,81.560,0.0000,-0.0000,1.0000
C01784=44.210,-116.910,81.560,0.0000,-0.0000,1.0000
C01785=36.970,-119.340,81.270,0.0000,-0.0000,1.0000
C01786=29.920,-120.240,80.840,-0.0000,-0.0400,1.0000
C01787=23.710,-117.990,80.410,-0.0500,-0.0700,1.0000
C01788=19.550,-113.090,79.890,-0.1300,-0.0600,0.9900
C01789=17.930,-106.340,78.890,-0.1300,-0.0300,0.9900
C01790=16.640,-99.090,76.890,-0.1100,-0.0200,0.9900
C01791=15.430,-92.670,74.320,-0.0600,-0.0100,1.0000
C01792=14.120,-87.910,71.850,0.0500,0.0200,1.0000
C01793=11.910,-85.200,70.080,0.2600,0.4200,0.8700
C01794=7.570,-84.630,69.380,0.0200,0.6200,0.7900
C01795=3.580,-84.830,69.350,-0.0300,0.6200,0.7800
C01796=0.000,-84.900,69.370,-0.0000,0.6200,0.7800
C01797=0.000,-84.900,69.370,-0.0000,0.6200,0.7800
C01798=-3.580,-84.830,69.350,0.0300,0.6200,0.7800
C01799=-7.570,-84.630,69.380,-0.0200,0.6200,0.7900
C01800=-11.910,-85.200,70.080,-0.2600,0.4200,0.8700
C01801=-14.120,-87.910,71.850,-0.0500,0.0200,1.0000
C01802=-15.430,-92.670,74.320,0.0600,-0.0100,1.0000
C01803=-16.640,-99.090,76.890,0.1100,-0.0200,0.9900
C01804=-17.930,-106.340,78.890,0.1300,-0.0300,0.9900
C01805=-19.550,-113.090,79.890,0.1300,-0.0600,0.9900
C01806=-23.710,-117.990,80.410,0.0500,-0.0700,1.0000
C01807=-29.920,-120.240,80.840,0.0000,-0.0400,1.0000
C01808=-36.970,-119.340,81.270,-0.0000,-0.0000,1.0000
C01809=-44.210,-116.910,81.560,-0.0000,-0.0000,1.0000
C01810=-51.410,-113.930,81.560,-0.0000,-0.0000,1.0000
C01811=-58.240,-110.530,81.270,-0.0000,-0.0000,1.0000
C01812=-63.870,-106.180,80.840,-0.0300,-0.0300,1.0000
C01813=-66.670,-100.190,80.410,-0.0800,-0.0200,1.0000
C01814=-66.140,-93.790,79.890,-0.1300,0.0500,0.9900
C01815=-62.520,-87.880,78.890,-0.1200,0.0700,0.9900
C01816=-58.300,-81.830,76.890,-0.0900,0.0600,0.9900
C01817=-54.620,-76.440,74.320,-0.0500,0.0300,1.0000
C01818=-52.180,-72.140,71.850,0.0500,-0.0200,1.0000
C01819=-51.830,-68.670,70.080,0.4700,0.1100,0.8700
C01820=-54.490,-65.200,69.380,0.4500,0.4200,0.7900
C01821=-57.450,-62.510,69.350,0.4200,0.4600,0.7800
C01822=-60.030,-60.030,69.370,0.4400,0.4400,0.7800
C01823=-62.510,-57.450,69.350,0.4600,0.4200,0.7800
C01824=-65.200,-54.490,69.380,0.4200,0.4500,0.7900
C01825=-68.670,-51.830,70.080,0.1100,0.4700,0.8700
C01826=-72.140,-52.180,71.850,-0.0200,0.0500,1.0000
C01827=-76.440,-54.620,74.320,0.0300,-0.0500,1.0000
C01828=-81.830,-58.300,76.890,0.0600,-0.0900,0.9900
C01829=-87.880,-62.520,78.890,0.0700,-0.1200,0.9900
C01830=-93.790,-66.140,79.890,0.0500,-0.1300,0.9900
C01831=-100.190,-66.670,80.410,-0.0200,-0.0800,1.0000
C01832=-106.180,-63.870,80.840,-0.0300,-0.0300,1.0000
C01833=-110.530,-58.240,81.270,-0.0000,-0.0000,1.0000
C01834=-113.930,-51.410,81.560,-0.0000,-0.0000,1.0000
C01835=-116.910,-44.210,81.560,-0.0000,-0.0000,1.0000
C01836=-119.340,-36.970,81.270,-0.0000,-0.0000,1.0000
C01837=-120.240,-29.920,80.840,-0.0400,0.0000,1.0000
C01838=-117.990,-23.710,80.410,-0.0700,0.0500,1.0000
C01839=-113.090,-19.550,79.890,-0.0600,0.1300,0.9900
C01840=-106.340,-17.930,78.890,-0.0300,0.1300,0.9900
C01841=-99.090,-16.640,76.890,-0.0200,0.1100,0.9900
C01842=-92.670,-15.430,74.320,-0.0100,0.0600,1.0000
C01843=-87.910,-14.120,71.850,0.0200,-0.0500,1.0000
C01844=-85.200,-11.910,70.080,0.4200,-0.2600,0.8700
C01845=-84.630,-7.570,69.380,0.6200,-0.0200,0.7900
C01846=-84.830,-3.580,69.350,0.6200,0.0300,0.7800
C01847=-84.900,0.000,69.370,0.6200,0.0000,0.7800
C01848=-84.830,3.580,69.350,0.6200,-0.0300,0.7800
C01849=-84.630,7.570,69.380,0.6200,0.0200,0.7900
C01850=-85.200,11.910,70.080,0.4200,0.2600,0.8700
C01851=-87.910,14.120,71.850,0.0200,0.0500,1.0000
C01852=-92.670,15.430,74.320,-0.0100,-0.0600,1.0000
C01853=-99.090,16.640,76.890,-0.0200,-0.1100,0.9900
C01854=-106.340,17.930,78.890,-0.0300,-0.1300,0.9900
C01855=-113.090,19.550,79.890,-0.0600,-0.1300,0.9900
C01856=-117.990,23.710,80.410,-0.0700,-0.0500,1.0000
C01857=-120.240,29.920,80.840,-0.0400,-0.0000,1.0000
C01858=-119.340,36.970,81.270,-0.0000,0.0000,1.0000
C01859=-116.910,44.210,81.560,-0.0000,0.0000,1.0000
C01860=-113.930,51.410,81.560,-0.0000,0.0000,1.0000
C01861=-110.530,58.240,81.270,-0.0000,0.0000,1.0000
C01862=-106.180,63.870,80.840,-0.0300,0.0300,1.0000
C01863=-100.190,66.670,80.410,-0.0200,0.0800,1.0000
C01864=-93.790,66.140,79.890,0.0500,0.1300,0.9900
C01865=-87.880,62.520,78.890,0.0700,0.1200,0.9900
C01866=-81.830,58.300,76.890,0.0600,0.0900,0.9900
C01867=-76.440,54.620,74.320,0.0300,0.0500,1.0000
C01868=-72.140,52.180,71.850,-0.0200,-0.0500,1.0000
C01869=-68.670,51.830,70.080,0.1100,-0.4700,0.8700
C01870=-65.200,54.490,69.380,0.4200,-0.4500,0.7900
C01871=-62.510,57.450,69.350,0.4600,-0.4200,0.7800
C01872=-60.030,60.030,69.370,0.4400,-0.4400,0.7800
C01873=-57.450,62.510,69.350,0.4200,-0.4600,0.7800
C01874=-54.490,65.200,69.380,0.4500,-0.4200,0.7900
C01875=-51.830,68.670,70.080,0.4700,-0.1100,0.8700
C01876=-52.180,72.140,71.850,0.0500,0.0200,1.0000
C01877=-54.620,76.440,74.320,-0.0500,-0.0300,1.0000
C01878=-58.300,81.830,76.890,-0.0900,-0.0600,0.9900
C01879=-62.520,87.880,78.890,-0.1200,-0.0700,0.9900
C01880=-66.140,93.790,79.890,-0.1300,-0.0500,0.9900
C01881=-66.670,100.190,80.410,-0.0800,0.0200,1.0000
C01882=-63.870,106.180,80.840,-0.0300,0.0300,1.0000
C01883=-58.240,110.530,81.270,-0.0000,0.0000,1.0000
C01884=-51.410,113.930,81.560,-0.0000,0.0000,1.0000
C01885=-44.210,116.910,81.560,-0.0000,0.0000,1.0000
C01886=-36.970,119.340,81.270,-0.0000,0.0000,1.0000
C01887=-29.920,120.240,80.840,0.0000,0.0400,1.0000
C01888=-23.710,117.990,80.410,0.0500,0.0700,1.0000
C01889=-19.550,113.090,79.890,0.1300,0.0600,0.9900
C01890=-17.930,106.340,78.890,0.1300,0.0300,0.9900
C01891=-16.640,99.090,76.890,0.1100,0.0200,0.9900
C01892=-15.430,92.670,74.320,0.0600,0.0100,1.0000
C01893=-14.120,87.910,71.850,-0.0500,-0.0200,1.0000
C01894=-11.910,85.200,70.080,-0.2600,-0.4200,0.8700
C01895=-7.570,84.630,69.380,-0.0200,-0.6200,0.7900
C01896=-3.580,84.830,69.350,0.0300,-0.6200,0.7800
C01897=0.000,84.900,69.370,-0.0000,-0.6200,0.7800
C01898=0.000,83.840,70.700,-0.0000,-0.6200,0.7800
C01899=-3.480,83.770,70.680,0.0300,-0.6200,0.7800
C01900=-7.410,83.590,70.710,-0.0200,-0.6100,0.7900
C01901=-11.710,84.200,71.430,-0.2600,-0.4000,0.8800
C01902=-13.880,86.990,73.260,-0.0400,-0.0100,1.0000
C01903=-15.150,91.900,75.810,0.0600,0.0100,1.0000
C01904=-16.340,98.510,78.470,0.1100,0.0200,0.9900
C01905=-17.620,105.970,80.520,0.1300,0.0300,0.9900
C01906=-19.220,112.910,81.540,0.1300,0.0600,0.9900
C01907=-23.390,117.950,82.080,0.0500,0.0700,1.0000
C01908=-29.670,120.290,82.520,0.0000,0.0400,1.0000
C01909=-36.820,119.400,82.970,-0.0000,0.0000,1.0000
C01910=-44.160,116.930,83.260,-0.0000,0.0000,1.0000
C01911=-51.460,113.910,83.260,-0.0000,0.0000,1.0000
C01912=-58.390,110.460,82.970,-0.0000,0.0000,1.0000
C01913=-64.070,106.040,82.520,-0.0300,0.0300,1.0000
C01914=-66.860,99.940,82.080,-0.0800,0.0200,1.0000
C01915=-66.250,93.430,81.540,-0.1300,-0.0500,0.9900
C01916=-62.480,87.390,80.520,-0.1200,-0.0700,0.9900
C01917=-58.100,81.210,78.470,-0.0900,-0.0600,0.9900
C01918=-54.270,75.700,75.810,-0.0500,-0.0300,1.0000
C01919=-51.700,71.330,73.260,0.0400,0.0200,1.0000
C01920=-51.260,67.810,71.430,0.4700,-0.1000,0.8800
C01921=-53.870,64.350,70.710,0.4500,-0.4200,0.7900
C01922=-56.780,61.700,70.680,0.4200,-0.4600,0.7800
C01923=-59.280,59.280,70.700,0.4400,-0.4400,0.7800
C01924=-61.700,56.780,70.680,0.4600,-0.4200,0.7800
C01925=-64.350,53.870,70.710,0.4200,-0.4500,0.7900
C01926=-67.810,51.260,71.430,0.1000,-0.4700,0.8800
C01927=-71.330,51.700,73.260,-0.0200,-0.0400,1.0000
C01928=-75.700,54.270,75.810,0.0300,0.0500,1.0000
C01929=-81.210,58.100,78.470,0.0600,0.0900,0.9900
C01930=-87.390,62.480,80.520,0.0700,0.1200,0.9900
C01931=-93.430,66.250,81.540,0.0500,0.1300,0.9900
C01932=-99.940,66.860,82.080,-0.0200,0.0800,1.0000
C01933=-106.040,64.070,82.520,-0.0300,0.0300,1.0000
C01934=-110.460,58.390,82.970,-0.0000,0.0000,1.0000
C01935=-113.910,51.460,83.260,-0.0000,0.0000,1.0000
C01936=-116.930,44.160,83.260,-0.0000,0.0000,1.0000
C01937=-119.400,36.820,82.970,-0.0000,0.0000,1.0000
C01938=-120.290,29.670,82.520,-0.0400,-0.0000,1.0000
C01939=-117.950,23.390,82.080,-0.0700,-0.0500,1.0000
C01940=-112.910,19.220,81.540,-0.0600,-0.1300,0.9900
C01941=-105.970,17.620,80.520,-0.0300,-0.1300,0.9900
